C07183=1025.011,-6.218,-95.865,167.267,47.387,158.718
C07184=1025.005,-6.466,-95.851,167.264,47.390,158.718
C07185=1024.999,-6.717,-95.837,167.261,47.393,158.718
C07186=1024.992,-6.966,-95.824,167.259,47.397,158.718
C07187=1024.987,-7.216,-95.810,167.256,47.400,158.718
C07188=1024.980,-7.465,-95.796,167.254,47.403,158.719
C07189=1024.974,-7.714,-95.782,167.250,47.406,158.719
C07190=1024.967,-7.964,-95.768,167.248,47.410,158.719
C07191=1024.962,-8.214,-95.754,167.245,47.413,158.719
C07192=1024.956,-8.463,-95.741,167.242,47.416,158.720
C07193=1024.949,-8.713,-95.726,167.240,47.419,158.720
C07194=1024.943,-8.962,-95.713,167.237,47.422,158.720
C07195=1024.938,-9.212,-95.699,167.234,47.425,158.720
C07196=1024.932,-9.461,-95.685,167.232,47.428,158.721
C07197=1024.925,-9.711,-95.671,167.228,47.431,158.721
C07198=1024.920,-9.961,-95.658,167.227,47.435,158.721
C07199=1024.913,-10.210,-95.644,167.223,47.438,158.721
C07200=1024.907,-10.460,-95.629,167.221,47.441,158.721
C07201=1024.901,-10.709,-95.616,167.218,47.444,158.722
C07202=1024.896,-10.959,-95.602,167.215,47.448,158.722
C07203=1024.889,-11.209,-95.589,167.213,47.451,158.722
C07204=1024.883,-11.458,-95.575,167.210,47.454,158.722
C07205=1024.877,-11.707,-95.561,167.208,47.457,158.723
C07206=1024.872,-11.957,-95.548,167.204,47.460,158.723
C07207=1024.865,-12.207,-95.534,167.201,47.464,158.723
C07208=1024.859,-12.457,-95.520,167.199,47.466,158.723
C07209=1024.853,-12.705,-95.506,167.196,47.470,158.723
C07210=1024.847,-12.955,-95.492,167.194,47.472,158.724
C07211=1024.841,-13.205,-95.479,167.191,47.476,158.724
C07212=1024.835,-13.454,-95.465,167.189,47.479,158.724
C07213=1024.829,-13.704,-95.451,167.186,47.482,158.724
C07214=1024.823,-13.953,-95.438,167.182,47.485,158.725
C07215=1024.817,-14.202,-95.424,167.180,47.488,158.725
C07216=1024.811,-14.453,-95.410,167.177,47.491,158.725
C07217=1024.805,-14.702,-95.397,167.175,47.494,158.725
C07218=1024.799,-14.952,-95.383,167.172,47.497,158.725
C07219=1024.793,-15.201,-95.370,167.169,47.501,158.726
C07220=1024.787,-15.451,-95.355,167.167,47.504,158.726
C07221=1024.781,-15.700,-95.342,167.163,47.507,158.726
C07222=1024.775,-15.950,-95.329,167.161,47.510,158.726
C07223=1024.770,-16.200,-95.316,167.158,47.514,158.727
C07224=1024.763,-16.449,-95.303,167.155,47.517,158.727
C07225=1024.757,-16.699,-95.289,167.153,47.520,158.727
C07226=1024.750,-16.948,-95.276,167.150,47.523,158.727
C07227=1024.744,-17.198,-95.262,167.147,47.527,158.727
C07228=1024.739,-17.447,-95.248,167.145,47.530,158.728
C07229=1024.733,-17.697,-95.236,167.141,47.533,158.728
C07230=1024.726,-17.947,-95.222,167.138,47.537,158.728
C07231=1024.720,-18.196,-95.209,167.136,47.539,158.728
C07232=1024.714,-18.446,-95.195,167.133,47.543,158.729
C07233=1024.708,-18.695,-95.182,167.130,47.546,158.729
C07234=1024.702,-18.945,-95.169,167.128,47.549,158.729
C07235=1024.696,-19.194,-95.156,167.125,47.552,158.729
C07236=1024.690,-19.444,-95.142,167.122,47.555,158.729
C07237=1024.684,-19.694,-95.129,167.120,47.559,158.730
C07238=1024.677,-19.943,-95.115,167.117,47.562,158.730
C07239=1024.671,-20.193,-95.103,167.114,47.565,158.730
C07240=1024.665,-20.473,-95.087,167.110,47.569,158.730
C07241=1024.658,-20.753,-95.073,167.107,47.572,158.731
C07242=1024.651,-21.034,-95.058,167.104,47.576,158.731
C07243=1024.645,-21.315,-95.043,167.101,47.580,158.731
C07244=1024.639,-21.564,-95.030,167.098,47.583,158.731
C07245=1024.633,-21.813,-95.017,167.096,47.586,158.732
C07246=1024.626,-22.063,-95.003,167.093,47.589,158.732
C07247=1024.620,-22.313,-94.990,167.091,47.592,158.732
C07248=1024.614,-22.562,-94.977,167.088,47.596,158.732
C07249=1024.608,-22.812,-94.963,167.085,47.599,158.732
C07250=1024.602,-23.062,-94.951,167.082,47.602,158.733
C07251=1024.596,-23.311,-94.937,167.079,47.605,158.733
C07252=1024.591,-23.560,-94.924,167.076,47.609,158.733
C07253=1024.585,-23.810,-94.911,167.074,47.612,158.733
C07254=1024.578,-24.060,-94.898,167.071,47.615,158.733
C07255=1024.572,-24.309,-94.885,167.068,47.618,158.734
C07256=1024.566,-24.559,-94.872,167.066,47.621,158.734
C07257=1024.560,-24.808,-94.859,167.062,47.624,158.734
C07258=1024.555,-25.058,-94.846,167.059,47.628,158.734
C07259=1024.549,-25.307,-94.832,167.057,47.631,158.735
C07260=1024.543,-25.557,-94.820,167.054,47.634,158.735
C07261=1024.537,-25.807,-94.806,167.051,47.637,158.735
C07262=1024.530,-26.056,-94.793,167.049,47.640,158.735
C07263=1024.525,-26.306,-94.780,167.046,47.643,158.735
C07264=1024.519,-26.555,-94.767,167.044,47.646,158.736
C07265=1024.513,-26.805,-94.754,167.040,47.650,158.736
C07266=1024.507,-27.054,-94.741,167.037,47.653,158.736
C07267=1024.501,-27.304,-94.728,167.035,47.656,158.736
C07268=1024.495,-27.554,-94.715,167.032,47.659,158.736
C07269=1024.489,-27.804,-94.703,167.029,47.663,158.737
C07270=1024.483,-28.053,-94.689,167.026,47.666,158.737
C07271=1024.477,-28.303,-94.677,167.024,47.669,158.737
C07272=1024.471,-28.553,-94.664,167.021,47.672,158.737
C07273=1024.465,-28.802,-94.651,167.018,47.676,158.737
C07274=1024.459,-29.052,-94.638,167.015,47.678,158.738
C07275=1024.452,-29.301,-94.625,167.012,47.682,158.738
C07276=1024.447,-29.551,-94.613,167.009,47.685,158.738
C07277=1024.441,-29.801,-94.600,167.006,47.689,158.738
C07278=1024.434,-30.050,-94.587,167.004,47.691,158.738
C07279=1024.429,-30.300,-94.574,167.001,47.695,158.739
C07280=1024.423,-30.550,-94.562,166.998,47.698,158.739
C07281=1024.416,-30.799,-94.549,166.995,47.702,158.739
C07282=1024.410,-31.049,-94.536,166.992,47.704,158.739
C07283=1024.404,-31.298,-94.524,166.990,47.708,158.740
C07284=1024.398,-31.547,-94.511,166.986,47.711,158.740
C07285=1024.392,-31.797,-94.498,166.984,47.714,158.740
C07286=1024.386,-32.047,-94.486,166.981,47.718,158.740
C07287=1024.380,-32.296,-94.473,166.978,47.721,158.740
C07288=1024.374,-32.546,-94.460,166.975,47.724,158.741
C07289=1024.368,-32.796,-94.447,166.973,47.727,158.741
C07290=1024.362,-33.046,-94.435,166.970,47.731,158.741
C07291=1024.356,-33.295,-94.422,166.967,47.734,158.741
C07292=1024.350,-33.545,-94.410,166.964,47.737,158.741
C07293=1024.344,-33.794,-94.397,166.961,47.740,158.742
C07294=1024.338,-34.044,-94.385,166.958,47.744,158.742
C07295=1024.332,-34.293,-94.372,166.955,47.747,158.742
C07296=1024.326,-34.543,-94.359,166.953,47.750,158.742
C07297=1024.320,-34.793,-94.347,166.950,47.753,158.742
C07298=1024.314,-35.043,-94.334,166.947,47.757,158.743
C07299=1024.308,-35.292,-94.321,166.945,47.760,158.743
C07300=1024.303,-35.541,-94.309,166.942,47.763,158.743
C07301=1024.296,-35.791,-94.297,166.938,47.766,158.743
C07302=1024.290,-36.040,-94.284,166.935,47.770,158.743
C07303=1024.284,-36.290,-94.271,166.933,47.772,158.744
C07304=1024.278,-36.570,-94.257,166.930,47.776,158.744
C07305=1024.272,-36.849,-94.243,166.926,47.780,158.744
C07306=1024.265,-37.129,-94.230,166.923,47.784,158.744
C07307=1024.258,-37.408,-94.215,166.920,47.787,158.745
C07308=1024.252,-37.658,-94.203,166.917,47.791,158.745
C07309=1024.246,-37.908,-94.190,166.915,47.793,158.745
C07310=1024.241,-38.157,-94.178,166.912,47.797,158.745
C07311=1024.234,-38.407,-94.166,166.908,47.800,158.745
C07312=1024.228,-38.656,-94.153,166.905,47.803,158.745
C07313=1024.222,-38.906,-94.140,166.903,47.807,158.746
C07314=1024.216,-39.156,-94.128,166.900,47.810,158.746
C07315=1024.211,-39.405,-94.115,166.897,47.813,158.746
C07316=1024.204,-39.654,-94.103,166.894,47.816,158.746
C07317=1024.198,-39.904,-94.091,166.892,47.820,158.747
C07318=1024.193,-40.155,-94.079,166.889,47.823,158.747
C07319=1024.187,-40.404,-94.067,166.886,47.826,158.747
C07320=1024.181,-40.654,-94.055,166.883,47.830,158.747
C07321=1024.175,-40.903,-94.042,166.880,47.833,158.747
C07322=1024.168,-41.153,-94.030,166.877,47.836,158.748
C07323=1024.163,-41.402,-94.018,166.874,47.840,158.748
C07324=1024.156,-41.652,-94.006,166.871,47.843,158.748
C07325=1024.151,-41.902,-93.994,166.868,47.846,158.748
C07326=1024.145,-42.152,-93.981,166.866,47.850,158.748
C07327=1024.139,-42.400,-93.969,166.863,47.853,158.749
C07328=1024.133,-42.650,-93.957,166.860,47.856,158.749
C07329=1024.126,-42.900,-93.946,166.857,47.859,158.749
C07330=1024.121,-43.150,-93.933,166.854,47.863,158.749
C07331=1024.115,-43.400,-93.921,166.852,47.866,158.749
C07332=1024.108,-43.649,-93.909,166.848,47.869,158.750
C07333=1024.103,-43.899,-93.896,166.845,47.873,158.750
C07334=1024.097,-44.148,-93.885,166.842,47.876,158.750
C07335=1024.091,-44.398,-93.872,166.839,47.879,158.750
C07336=1024.085,-44.648,-93.860,166.837,47.882,158.750
C07337=1024.079,-44.897,-93.849,166.834,47.886,158.751
C07338=1024.073,-45.147,-93.836,166.831,47.889,158.751
C07339=1024.067,-45.396,-93.825,166.828,47.892,158.751
C07340=1024.061,-45.646,-93.812,166.825,47.895,158.751
C07341=1024.055,-45.896,-93.800,166.823,47.899,158.751
C07342=1024.049,-46.145,-93.789,166.819,47.902,158.752
C07343=1024.044,-46.395,-93.776,166.816,47.905,158.752
C07344=1024.037,-46.645,-93.764,166.813,47.909,158.752
C07345=1024.032,-46.894,-93.753,166.811,47.912,158.752
C07346=1024.026,-47.144,-93.740,166.808,47.915,158.752
C07347=1024.020,-47.393,-93.729,166.805,47.918,158.753
C07348=1024.014,-47.643,-93.716,166.802,47.922,158.753
C07349=1024.008,-47.893,-93.705,166.799,47.925,158.753
C07350=1024.002,-48.142,-93.693,166.797,47.928,158.753
C07351=1023.996,-48.392,-93.680,166.793,47.932,158.753
C07352=1023.991,-48.642,-93.669,166.790,47.935,158.753
C07353=1023.985,-48.892,-93.657,166.787,47.938,158.754
C07354=1023.978,-49.141,-93.645,166.785,47.941,158.754
C07355=1023.973,-49.391,-93.633,166.782,47.945,158.754
C07356=1023.967,-49.641,-93.621,166.779,47.948,158.754
C07357=1023.961,-49.890,-93.609,166.776,47.951,158.754
C07358=1023.956,-50.140,-93.597,166.773,47.954,158.755
C07359=1023.950,-50.389,-93.586,166.770,47.957,158.755
C07360=1023.944,-50.639,-93.573,166.767,47.961,158.755
C07361=1023.938,-50.889,-93.562,166.764,47.964,158.755
C07362=1023.931,-51.138,-93.550,166.761,47.967,158.755
C07363=1023.926,-51.389,-93.538,166.758,47.971,158.756
C07364=1023.920,-51.637,-93.527,166.755,47.974,158.756
C07365=1023.913,-51.888,-93.516,166.753,47.978,158.756
C07366=1023.908,-52.137,-93.505,166.750,47.981,158.756
C07367=1023.901,-52.387,-93.493,166.747,47.984,158.756
C07368=1023.894,-52.666,-93.480,166.743,47.988,158.757
C07369=1023.887,-52.947,-93.467,166.740,47.992,158.757
C07370=1023.881,-53.227,-93.454,166.737,47.996,158.757
C07371=1023.875,-53.507,-93.441,166.733,48.000,158.757
C07372=1023.869,-53.756,-93.430,166.730,48.004,158.757
C07373=1023.862,-54.006,-93.418,166.727,48.007,158.758
C07374=1023.856,-54.255,-93.407,166.725,48.010,158.758
C07375=1023.850,-54.505,-93.395,166.722,48.013,158.758
C07376=1023.844,-54.755,-93.385,166.719,48.017,158.758
C07377=1023.838,-55.005,-93.372,166.716,48.021,158.759
C07378=1023.833,-55.254,-93.361,166.713,48.024,158.759
C07379=1023.826,-55.504,-93.350,166.710,48.028,158.759
C07380=1023.820,-55.753,-93.338,166.706,48.031,158.759
C07381=1023.814,-56.003,-93.327,166.704,48.035,158.759
C07382=1023.809,-56.253,-93.316,166.700,48.038,158.760
C07383=1023.803,-56.502,-93.304,166.698,48.041,158.760
C07384=1023.796,-56.752,-93.293,166.695,48.045,158.760
C07385=1023.791,-57.002,-93.282,166.692,48.048,158.760
C07386=1023.784,-57.251,-93.270,166.689,48.052,158.760
C07387=1023.778,-57.501,-93.259,166.686,48.055,158.761
C07388=1023.773,-57.751,-93.247,166.683,48.058,158.761
C07389=1023.767,-58.001,-93.236,166.680,48.062,158.761
C07390=1023.761,-58.250,-93.225,166.677,48.065,158.761
C07391=1023.755,-58.500,-93.213,166.674,48.068,158.761
C07392=1023.749,-58.749,-93.203,166.672,48.072,158.762
C07393=1023.742,-58.999,-93.191,166.669,48.075,158.762
C07394=1023.737,-59.249,-93.180,166.666,48.079,158.762
C07395=1023.731,-59.498,-93.168,166.663,48.082,158.762
C07396=1023.725,-59.748,-93.157,166.659,48.085,158.762
C07397=1023.719,-59.998,-93.146,166.656,48.089,158.763
C07398=1023.714,-60.247,-93.135,166.653,48.092,158.763
C07399=1023.707,-60.497,-93.124,166.650,48.096,158.763
C07400=1023.701,-60.746,-93.112,166.647,48.099,158.763
C07401=1023.696,-60.996,-93.101,166.645,48.102,158.763
C07402=1023.690,-61.246,-93.090,166.642,48.106,158.764
C07403=1023.684,-61.496,-93.079,166.639,48.109,158.764
C07404=1023.678,-61.745,-93.068,166.636,48.113,158.764
C07405=1023.672,-61.995,-93.057,166.633,48.116,158.764
C07406=1023.666,-62.245,-93.046,166.629,48.119,158.764
C07407=1023.660,-62.494,-93.034,166.627,48.123,158.764
C07408=1023.655,-62.744,-93.022,166.623,48.126,158.765
///RCONF 1,0,0,1,0,0,0,0,0,0,0,0,0,0,0,0,0,0,0,0,0,0,0,0
C07409=1023.649,-62.994,-93.012,166.620,48.129,158.765
C07410=1023.643,-63.243,-93.001,166.618,48.133,158.765
C07411=1023.637,-63.494,-92.989,166.615,48.136,158.765
C07412=1023.631,-63.743,-92.979,166.612,48.139,158.765
C07413=1023.625,-63.992,-92.968,166.609,48.143,158.765
C07414=1023.620,-64.242,-92.957,166.606,48.146,158.766
C07415=1023.614,-64.492,-92.945,166.603,48.150,158.766
C07416=1023.608,-64.742,-92.934,166.600,48.153,158.766
C07417=1023.603,-64.991,-92.923,166.596,48.156,158.766
C07418=1023.597,-65.241,-92.912,166.595,48.160,158.767
C07419=1023.590,-65.491,-92.901,166.591,48.163,158.767
C07420=1023.585,-65.741,-92.890,166.588,48.166,158.767
C07421=1023.579,-65.990,-92.879,166.585,48.169,158.767
C07422=1023.573,-66.240,-92.868,166.582,48.173,158.767
C07423=1023.568,-66.489,-92.857,166.579,48.176,158.767
C07424=1023.562,-66.740,-92.846,166.576,48.180,158.767
C07425=1023.556,-66.989,-92.835,166.573,48.183,158.768
C07426=1023.550,-67.239,-92.824,166.571,48.186,158.768
C07427=1023.545,-67.488,-92.813,166.568,48.190,158.768
C07428=1023.539,-67.738,-92.802,166.564,48.193,158.768
C07429=1023.533,-67.988,-92.791,166.561,48.196,158.768
C07430=1023.527,-68.237,-92.780,166.558,48.200,158.769
C07431=1023.521,-68.487,-92.769,166.555,48.203,158.769
C07432=1023.516,-68.768,-92.757,166.552,48.206,158.769
C07433=1023.508,-69.049,-92.744,166.549,48.210,158.769
C07434=1023.502,-69.330,-92.733,166.545,48.214,158.769
C07435=1023.496,-69.612,-92.720,166.542,48.218,158.769
C07436=1023.490,-69.861,-92.709,166.539,48.221,158.770
C07437=1023.484,-70.111,-92.698,166.536,48.225,158.770
C07438=1023.479,-70.360,-92.687,166.533,48.228,158.770
C07439=1023.473,-70.610,-92.676,166.530,48.231,158.770
C07440=1023.467,-70.859,-92.666,166.528,48.234,158.770
C07441=1023.462,-71.109,-92.655,166.524,48.237,158.770
C07442=1023.456,-71.359,-92.644,166.522,48.241,158.771
C07443=1023.450,-71.609,-92.633,166.518,48.244,158.771
C07444=1023.444,-71.859,-92.622,166.515,48.247,158.771
C07445=1023.439,-72.108,-92.611,166.512,48.251,158.771
C07446=1023.433,-72.358,-92.600,166.509,48.254,158.771
C07447=1023.428,-72.608,-92.590,166.506,48.257,158.771
C07448=1023.422,-72.858,-92.579,166.504,48.261,158.772
C07449=1023.416,-73.107,-92.568,166.501,48.264,158.772
C07450=1023.411,-73.356,-92.557,166.497,48.267,158.772
C07451=1023.405,-73.606,-92.546,166.494,48.270,158.772
C07452=1023.399,-73.856,-92.536,166.491,48.274,158.772
C07453=1023.394,-74.106,-92.525,166.488,48.277,158.772
C07454=1023.388,-74.355,-92.514,166.485,48.281,158.773
C07455=1023.383,-74.605,-92.504,166.483,48.284,158.773
C07456=1023.377,-74.855,-92.493,166.480,48.287,158.773
C07457=1023.371,-75.105,-92.483,166.477,48.291,158.773
C07458=1023.365,-75.355,-92.472,166.474,48.294,158.773
C07459=1023.359,-75.604,-92.462,166.470,48.297,158.773
C07460=1023.353,-75.854,-92.452,166.468,48.301,158.774
C07461=1023.347,-76.104,-92.441,166.464,48.304,158.774
C07462=1023.342,-76.354,-92.431,166.461,48.307,158.774
C07463=1023.336,-76.603,-92.420,166.458,48.311,158.774
C07464=1023.330,-76.853,-92.410,166.455,48.315,158.774
C07465=1023.324,-77.103,-92.399,166.452,48.318,158.774
C07466=1023.319,-77.353,-92.389,166.449,48.322,158.775
C07467=1023.313,-77.602,-92.378,166.446,48.325,158.775
C07468=1023.307,-77.852,-92.369,166.443,48.328,158.775
C07469=1023.301,-78.102,-92.358,166.440,48.332,158.775
C07470=1023.296,-78.352,-92.348,166.437,48.335,158.775
C07471=1023.290,-78.601,-92.337,166.434,48.338,158.775
C07472=1023.285,-78.851,-92.327,166.431,48.342,158.776
C07473=1023.279,-79.100,-92.317,166.429,48.345,158.776
C07474=1023.273,-79.350,-92.306,166.425,48.349,158.776
C07475=1023.268,-79.599,-92.296,166.422,48.352,158.776
C07476=1023.262,-79.849,-92.285,166.419,48.356,158.776
C07477=1023.256,-80.099,-92.275,166.416,48.359,158.777
C07478=1023.250,-80.349,-92.265,166.413,48.362,158.777
C07479=1023.245,-80.599,-92.255,166.410,48.366,158.777
C07480=1023.238,-80.848,-92.244,166.407,48.369,158.777
C07481=1023.233,-81.098,-92.234,166.404,48.373,158.777
C07482=1023.227,-81.348,-92.225,166.401,48.376,158.777
C07483=1023.221,-81.597,-92.214,166.398,48.380,158.778
C07484=1023.215,-81.847,-92.204,166.395,48.383,158.778
C07485=1023.209,-82.097,-92.194,166.392,48.387,158.778
C07486=1023.203,-82.347,-92.185,166.389,48.391,158.778
C07487=1023.197,-82.597,-92.174,166.386,48.395,158.779
C07488=1023.192,-82.846,-92.165,166.383,48.398,158.779
C07489=1023.186,-83.096,-92.154,166.380,48.402,158.779
C07490=1023.180,-83.346,-92.145,166.377,48.405,158.779
C07491=1023.175,-83.595,-92.134,166.374,48.408,158.779
C07492=1023.168,-83.845,-92.124,166.371,48.412,158.779
C07493=1023.163,-84.095,-92.114,166.368,48.415,158.780
C07494=1023.157,-84.345,-92.105,166.365,48.419,158.780
C07495=1023.151,-84.595,-92.094,166.362,48.422,158.780
C07496=1023.145,-84.877,-92.083,166.358,48.427,158.780
C07497=1023.138,-85.161,-92.072,166.354,48.431,158.780
C07498=1023.132,-85.443,-92.060,166.351,48.435,158.781
C07499=1023.125,-85.727,-92.049,166.347,48.439,158.781
C07500=1023.119,-85.977,-92.040,166.344,48.442,158.781
C07501=1023.114,-86.227,-92.030,166.341,48.446,158.781
C07502=1023.108,-86.476,-92.020,166.338,48.449,158.781
C07503=1023.103,-86.726,-92.010,166.335,48.453,158.781
C07504=1023.096,-86.975,-92.000,166.332,48.457,158.782
C07505=1023.091,-87.225,-91.990,166.329,48.460,158.782
C07506=1023.084,-87.475,-91.980,166.326,48.464,158.782
C07507=1023.080,-87.725,-91.970,166.323,48.467,158.782
C07508=1023.073,-87.974,-91.961,166.320,48.470,158.782
C07509=1023.068,-88.225,-91.951,166.317,48.474,158.783
C07510=1023.062,-88.474,-91.941,166.314,48.477,158.783
C07511=1023.057,-88.724,-91.931,166.311,48.481,158.783
C07512=1023.051,-88.974,-91.922,166.307,48.484,158.783
C07513=1023.045,-89.224,-91.912,166.304,48.488,158.783
C07514=1023.039,-89.473,-91.902,166.301,48.492,158.783
C07515=1023.034,-89.723,-91.892,166.298,48.495,158.784
C07516=1023.028,-89.973,-91.883,166.295,48.498,158.784
C07517=1023.023,-90.223,-91.872,166.292,48.502,158.784
C07518=1023.017,-90.472,-91.863,166.289,48.505,158.784
C07519=1023.012,-90.722,-91.853,166.286,48.509,158.784
C07520=1023.006,-90.972,-91.844,166.283,48.512,158.784
C07521=1022.999,-91.222,-91.834,166.280,48.516,158.784
C07522=1022.995,-91.471,-91.824,166.277,48.520,158.785
C07523=1022.988,-91.721,-91.815,166.274,48.523,158.785
C07524=1022.983,-91.971,-91.804,166.271,48.526,158.785
C07525=1022.977,-92.220,-91.795,166.269,48.530,158.785
C07526=1022.972,-92.470,-91.785,166.266,48.533,158.785
C07527=1022.966,-92.720,-91.776,166.263,48.536,158.786
C07528=1022.961,-92.969,-91.766,166.260,48.540,158.786
C07529=1022.955,-93.219,-91.756,166.257,48.543,158.786
C07530=1022.949,-93.469,-91.746,166.253,48.547,158.786
C07531=1022.944,-93.718,-91.737,166.251,48.551,158.786
C07532=1022.938,-93.969,-91.728,166.247,48.554,158.786
C07533=1022.933,-94.218,-91.718,166.244,48.557,158.787
C07534=1022.927,-94.468,-91.709,166.241,48.561,158.787
C07535=1022.922,-94.718,-91.698,166.238,48.564,158.787
C07536=1022.916,-94.967,-91.689,166.235,48.567,158.787
C07537=1022.911,-95.217,-91.679,166.232,48.571,158.787
C07538=1022.905,-95.466,-91.670,166.229,48.575,158.787
C07539=1022.900,-95.717,-91.660,166.226,48.578,158.787
C07540=1022.894,-95.967,-91.651,166.223,48.582,158.788
C07541=1022.888,-96.216,-91.642,166.220,48.585,158.788
C07542=1022.883,-96.466,-91.631,166.217,48.588,158.788
C07543=1022.877,-96.715,-91.622,166.213,48.591,158.788
C07544=1022.872,-96.966,-91.613,166.211,48.595,158.788
C07545=1022.866,-97.215,-91.604,166.207,48.599,158.788
C07546=1022.861,-97.465,-91.593,166.204,48.602,158.789
C07547=1022.855,-97.714,-91.584,166.201,48.606,158.789
C07548=1022.850,-97.965,-91.575,166.198,48.609,158.789
C07549=1022.843,-98.214,-91.566,166.195,48.612,158.789
C07550=1022.839,-98.464,-91.556,166.192,48.616,158.789
C07551=1022.833,-98.714,-91.547,166.189,48.620,158.789
C07552=1022.827,-98.963,-91.538,166.186,48.623,158.790
C07553=1022.821,-99.213,-91.528,166.183,48.627,158.790
C07554=1022.816,-99.463,-91.520,166.180,48.631,158.790
C07555=1022.809,-99.713,-91.510,166.177,48.634,158.790
C07556=1022.805,-99.963,-91.501,166.174,48.638,158.790
C07557=1022.799,-100.212,-91.492,166.171,48.641,158.791
C07558=1022.793,-100.462,-91.483,166.168,48.645,158.791
C07559=1022.787,-100.712,-91.474,166.165,48.648,158.791
C07560=1022.781,-100.997,-91.462,166.161,48.653,158.791
C07561=1022.775,-101.282,-91.453,166.157,48.657,158.791
C07562=1022.769,-101.568,-91.442,166.154,48.661,158.791
C07563=1022.761,-101.853,-91.432,166.151,48.665,158.792
C07564=1022.757,-102.103,-91.423,166.147,48.668,158.792
C07565=1022.751,-102.353,-91.413,166.145,48.672,158.792
C07566=1022.745,-102.602,-91.405,166.141,48.675,158.792
C07567=1022.739,-102.852,-91.395,166.139,48.679,158.792
C07568=1022.734,-103.102,-91.387,166.135,48.683,158.792
C07569=1022.728,-103.351,-91.377,166.132,48.686,158.793
C07570=1022.723,-103.602,-91.369,166.129,48.690,158.793
C07571=1022.718,-103.851,-91.359,166.126,48.693,158.793
C07572=1022.712,-104.101,-91.350,166.123,48.697,158.793
C07573=1022.706,-104.350,-91.341,166.120,48.700,158.793
C07574=1022.701,-104.600,-91.332,166.117,48.704,158.794
C07575=1022.695,-104.850,-91.323,166.114,48.708,158.794
C07576=1022.690,-105.100,-91.314,166.111,48.711,158.794
C07577=1022.684,-105.350,-91.305,166.108,48.715,158.794
C07578=1022.678,-105.599,-91.296,166.105,48.718,158.794
C07579=1022.673,-105.849,-91.288,166.102,48.722,158.794
C07580=1022.667,-106.099,-91.277,166.099,48.725,158.795
C07581=1022.662,-106.349,-91.269,166.096,48.729,158.795
C07582=1022.656,-106.599,-91.260,166.093,48.732,158.795
C07583=1022.651,-106.848,-91.251,166.089,48.736,158.795
C07584=1022.646,-107.098,-91.242,166.086,48.740,158.795
C07585=1022.640,-107.348,-91.234,166.083,48.743,158.795
C07586=1022.634,-107.598,-91.225,166.080,48.747,158.795
C07587=1022.629,-107.847,-91.216,166.077,48.750,158.796
C07588=1022.623,-108.098,-91.207,166.074,48.754,158.796
C07589=1022.618,-108.347,-91.199,166.071,48.758,158.796
C07590=1022.612,-108.596,-91.189,166.068,48.762,158.796
C07591=1022.606,-108.847,-91.181,166.065,48.765,158.796
C07592=1022.601,-109.097,-91.172,166.062,48.769,158.797
C07593=1022.596,-109.346,-91.164,166.059,48.772,158.797
C07594=1022.590,-109.597,-91.155,166.056,48.776,158.797
C07595=1022.584,-109.845,-91.146,166.053,48.779,158.797
C07596=1022.578,-110.095,-91.138,166.050,48.783,158.797
C07597=1022.573,-110.345,-91.129,166.047,48.787,158.797
C07598=1022.567,-110.595,-91.120,166.044,48.791,158.798
C07599=1022.562,-110.845,-91.112,166.041,48.794,158.798
C07600=1022.557,-111.095,-91.103,166.038,48.798,158.798
C07601=1022.550,-111.345,-91.094,166.034,48.801,158.798
C07602=1022.545,-111.594,-91.085,166.031,48.805,158.798
C07603=1022.540,-111.844,-91.077,166.028,48.809,158.798
C07604=1022.535,-112.094,-91.068,166.025,48.812,158.799
C07605=1022.529,-112.344,-91.059,166.022,48.816,158.799
C07606=1022.524,-112.594,-91.051,166.019,48.820,158.799
C07607=1022.518,-112.844,-91.042,166.016,48.823,158.799
C07608=1022.512,-113.093,-91.035,166.013,48.827,158.799
C07609=1022.507,-113.343,-91.026,166.010,48.830,158.799
C07610=1022.501,-113.592,-91.017,166.007,48.834,158.800
C07611=1022.496,-113.842,-91.008,166.004,48.837,158.800
C07612=1022.490,-114.092,-91.000,166.001,48.841,158.800
C07613=1022.485,-114.342,-90.991,165.998,48.845,158.800
C07614=1022.480,-114.591,-90.983,165.995,48.848,158.800
C07615=1022.474,-114.842,-90.974,165.992,48.852,158.800
C07616=1022.468,-115.091,-90.966,165.989,48.855,158.801
C07617=1022.463,-115.341,-90.957,165.986,48.859,158.801
C07618=1022.457,-115.591,-90.949,165.983,48.863,158.801
C07619=1022.452,-115.840,-90.940,165.979,48.867,158.801
C07620=1022.447,-116.091,-90.933,165.976,48.871,158.801
C07621=1022.441,-116.341,-90.924,165.973,48.874,158.801
C07622=1022.435,-116.590,-90.916,165.970,48.878,158.802
C07623=1022.430,-116.840,-90.907,165.967,48.881,158.802
C07624=1022.424,-117.125,-90.898,165.964,48.885,158.802
C07625=1022.418,-117.410,-90.888,165.960,48.889,158.802
C07626=1022.411,-117.695,-90.879,165.956,48.894,158.802
C07627=1022.405,-117.980,-90.869,165.953,48.898,158.803
C07628=1022.400,-118.229,-90.861,165.951,48.902,158.803
C07629=1022.394,-118.480,-90.853,165.946,48.905,158.803
C07630=1022.388,-118.730,-90.845,165.944,48.909,158.803
C07631=1022.383,-118.980,-90.836,165.940,48.913,158.803
C07632=1022.378,-119.229,-90.828,165.938,48.917,158.803
C07633=1022.372,-119.479,-90.819,165.934,48.920,158.804
C07634=1022.366,-119.728,-90.811,165.932,48.924,158.804
C07635=1022.361,-119.979,-90.804,165.928,48.927,158.804
C07636=1022.356,-120.228,-90.795,165.926,48.931,158.804
C07637=1022.350,-120.478,-90.787,165.922,48.934,158.804
C07638=1022.345,-120.727,-90.779,165.920,48.938,158.804
C07639=1022.340,-120.977,-90.770,165.917,48.942,158.805
C07640=1022.335,-121.228,-90.762,165.914,48.946,158.805
C07641=1022.329,-121.477,-90.755,165.911,48.950,158.805
C07642=1022.323,-121.727,-90.746,165.908,48.953,158.805
C07643=1022.318,-121.977,-90.738,165.905,48.957,158.805
C07644=1022.312,-122.226,-90.730,165.902,48.960,158.806
C07645=1022.307,-122.476,-90.722,165.898,48.964,158.806
C07646=1022.302,-122.726,-90.713,165.895,48.968,158.806
C07647=1022.296,-122.976,-90.706,165.892,48.972,158.806
C07648=1022.291,-123.226,-90.698,165.889,48.975,158.806
C07649=1022.286,-123.475,-90.689,165.886,48.979,158.806
C07650=1022.280,-123.725,-90.682,165.883,48.982,158.806
C07651=1022.275,-123.975,-90.674,165.880,48.986,158.807
C07652=1022.269,-124.225,-90.665,165.877,48.989,158.807
C07653=1022.264,-124.475,-90.658,165.874,48.993,158.807
C07654=1022.259,-124.724,-90.650,165.871,48.997,158.807
C07655=1022.253,-124.975,-90.642,165.868,49.001,158.807
C07656=1022.248,-125.224,-90.634,165.865,49.004,158.807
C07657=1022.242,-125.474,-90.625,165.862,49.008,158.808
C07658=1022.237,-125.724,-90.618,165.859,49.012,158.808
C07659=1022.231,-125.974,-90.610,165.855,49.016,158.808
C07660=1022.226,-126.224,-90.603,165.852,49.020,158.808
C07661=1022.220,-126.473,-90.594,165.849,49.023,158.808
C07662=1022.215,-126.723,-90.587,165.846,49.027,158.809
C07663=1022.209,-126.973,-90.578,165.843,49.031,158.809
C07664=1022.204,-127.223,-90.571,165.840,49.034,158.809
C07665=1022.198,-127.473,-90.563,165.837,49.038,158.809
C07666=1022.193,-127.723,-90.556,165.834,49.041,158.809
C07667=1022.188,-127.972,-90.547,165.831,49.045,158.809
C07668=1022.183,-128.222,-90.539,165.828,49.049,158.810
C07669=1022.178,-128.471,-90.531,165.825,49.051,158.809
C07670=1022.174,-128.721,-90.521,165.822,49.054,158.809
C07671=1022.170,-128.971,-90.511,165.820,49.056,158.809
C07672=1022.168,-129.220,-90.500,165.817,49.057,158.809
C07673=1022.165,-129.469,-90.490,165.815,49.058,158.809
C07674=1022.163,-129.719,-90.478,165.812,49.058,158.809
C07675=1022.161,-129.969,-90.465,165.809,49.058,158.808
C07676=1022.160,-130.219,-90.453,165.807,49.057,158.808
C07677=1022.160,-130.469,-90.439,165.805,49.056,158.807
C07678=1022.159,-130.719,-90.425,165.803,49.054,158.807
C07679=1022.160,-130.968,-90.410,165.801,49.052,158.806
C07680=1022.160,-131.219,-90.396,165.798,49.050,158.805
C07681=1022.162,-131.469,-90.379,165.797,49.046,158.804
C07682=1022.164,-131.718,-90.363,165.795,49.042,158.803
C07683=1022.166,-131.967,-90.346,165.793,49.038,158.802
C07684=1022.170,-132.218,-90.329,165.792,49.033,158.801
///RCONF 1,0,0,0,0,0,0,0,0,0,0,0,0,0,0,0,0,0,0,0,0,0,0,0
C07685=1022.172,-132.467,-90.310,165.790,49.028,158.800
C07686=1022.177,-132.717,-90.292,165.788,49.022,158.799
C07687=1022.181,-132.966,-90.273,165.786,49.016,158.798
C07688=1021.894,-132.993,-90.621,165.740,49.314,158.841
C07689=1021.889,-132.743,-90.640,165.742,49.320,158.842
C07690=1021.885,-132.493,-90.660,165.743,49.325,158.843
C07691=1021.882,-132.243,-90.677,165.744,49.331,158.845
C07692=1021.880,-131.993,-90.695,165.746,49.336,158.846
C07693=1021.877,-131.744,-90.712,165.748,49.340,158.847
C07694=1021.875,-131.494,-90.728,165.750,49.344,158.848
C07695=1021.874,-131.244,-90.744,165.752,49.346,158.848
C07696=1021.873,-130.994,-90.760,165.753,49.349,158.849
C07697=1021.873,-130.744,-90.775,165.756,49.352,158.850
C07698=1021.872,-130.495,-90.788,165.758,49.354,158.850
C07699=1021.874,-130.245,-90.801,165.761,49.355,158.851
C07700=1021.874,-129.995,-90.815,165.763,49.355,158.851
C07701=1021.876,-129.746,-90.827,165.765,49.355,158.852
C07702=1021.878,-129.496,-90.838,165.768,49.355,158.852
C07703=1021.880,-129.246,-90.849,165.770,49.355,158.852
C07704=1021.883,-128.996,-90.860,165.773,49.353,158.853
C07705=1021.887,-128.747,-90.870,165.775,49.351,158.853
C07706=1021.891,-128.497,-90.880,165.779,49.349,158.853
C07707=1021.895,-128.248,-90.888,165.781,49.346,158.853
C07708=1021.901,-127.998,-90.897,165.784,49.342,158.853
C07709=1021.905,-127.748,-90.905,165.787,49.339,158.853
C07710=1021.911,-127.499,-90.912,165.790,49.335,158.852
C07711=1021.916,-127.249,-90.920,165.793,49.331,158.852
C07712=1021.922,-127.000,-90.928,165.797,49.328,158.852
C07713=1021.927,-126.749,-90.935,165.800,49.323,158.852
C07714=1021.933,-126.500,-90.943,165.803,49.319,158.852
C07715=1021.938,-126.250,-90.951,165.806,49.316,158.852
C07716=1021.944,-126.000,-90.959,165.809,49.312,158.851
C07717=1021.949,-125.750,-90.967,165.812,49.309,158.851
C07718=1021.955,-125.500,-90.975,165.815,49.305,158.851
C07719=1021.960,-125.250,-90.982,165.817,49.301,158.851
C07720=1021.966,-125.001,-90.990,165.821,49.297,158.851
C07721=1021.971,-124.750,-90.998,165.824,49.293,158.850
C07722=1021.977,-124.501,-91.006,165.827,49.289,158.850
C07723=1021.981,-124.252,-91.014,165.830,49.286,158.850
C07724=1021.986,-124.002,-91.022,165.833,49.282,158.850
C07725=1021.992,-123.752,-91.030,165.836,49.278,158.850
C07726=1021.997,-123.502,-91.038,165.839,49.274,158.850
C07727=1022.003,-123.252,-91.046,165.842,49.271,158.849
C07728=1022.009,-123.003,-91.054,165.845,49.267,158.849
C07729=1022.013,-122.752,-91.062,165.848,49.263,158.849
C07730=1022.019,-122.503,-91.070,165.852,49.260,158.849
C07731=1022.025,-122.253,-91.078,165.855,49.256,158.849
C07732=1022.030,-122.003,-91.086,165.858,49.252,158.849
C07733=1022.035,-121.753,-91.094,165.861,49.248,158.848
C07734=1022.040,-121.503,-91.103,165.864,49.245,158.848
C07735=1022.046,-121.254,-91.111,165.867,49.241,158.848
C07736=1022.051,-121.004,-91.118,165.869,49.237,158.848
C07737=1022.056,-120.754,-91.127,165.872,49.234,158.848
C07738=1022.062,-120.505,-91.135,165.875,49.230,158.847
C07739=1022.068,-120.255,-91.143,165.878,49.226,158.847
C07740=1022.073,-120.005,-91.151,165.882,49.222,158.847
C07741=1022.079,-119.754,-91.159,165.885,49.219,158.847
C07742=1022.085,-119.505,-91.168,165.888,49.215,158.847
C07743=1022.090,-119.255,-91.176,165.891,49.211,158.847
C07744=1022.095,-119.005,-91.184,165.894,49.207,158.847
C07745=1022.101,-118.755,-91.192,165.897,49.203,158.846
C07746=1022.106,-118.506,-91.200,165.900,49.200,158.846
C07747=1022.111,-118.256,-91.209,165.903,49.196,158.846
C07748=1022.117,-118.006,-91.217,165.906,49.192,158.846
C07749=1022.123,-117.721,-91.227,165.910,49.188,158.846
C07750=1022.129,-117.436,-91.236,165.913,49.183,158.845
C07751=1022.135,-117.151,-91.245,165.916,49.179,158.845
C07752=1022.141,-116.866,-91.255,165.920,49.175,158.845
C07753=1022.147,-116.617,-91.263,165.923,49.172,158.845
C07754=1022.153,-116.367,-91.271,165.926,49.168,158.845
C07755=1022.158,-116.117,-91.280,165.929,49.164,158.844
C07756=1022.164,-115.867,-91.289,165.933,49.160,158.844
C07757=1022.169,-115.617,-91.297,165.936,49.156,158.844
C07758=1022.175,-115.368,-91.305,165.939,49.153,158.844
C07759=1022.180,-115.118,-91.313,165.942,49.149,158.844
C07760=1022.185,-114.868,-91.322,165.945,49.146,158.844
C07761=1022.191,-114.619,-91.330,165.948,49.142,158.843
C07762=1022.197,-114.368,-91.339,165.950,49.138,158.843
C07763=1022.203,-114.119,-91.347,165.954,49.134,158.843
C07764=1022.208,-113.869,-91.356,165.956,49.130,158.843
C07765=1022.213,-113.619,-91.364,165.961,49.127,158.843
C07766=1022.218,-113.370,-91.373,165.963,49.123,158.843
C07767=1022.224,-113.119,-91.381,165.967,49.119,158.843
C07768=1022.230,-112.869,-91.390,165.969,49.115,158.842
C07769=1022.235,-112.620,-91.398,165.973,49.112,158.842
C07770=1022.240,-112.370,-91.407,165.975,49.108,158.842
C07771=1022.245,-112.120,-91.415,165.978,49.105,158.842
C07772=1022.251,-111.870,-91.424,165.981,49.101,158.842
C07773=1022.256,-111.620,-91.433,165.984,49.098,158.841
C07774=1022.262,-111.370,-91.441,165.987,49.094,158.841
C07775=1022.268,-111.121,-91.449,165.990,49.090,158.841
C07776=1022.274,-110.871,-91.459,165.994,49.086,158.841
C07777=1022.279,-110.622,-91.467,165.997,49.082,158.841
C07778=1022.284,-110.372,-91.476,166.000,49.079,158.841
C07779=1022.290,-110.122,-91.484,166.003,49.075,158.840
C07780=1022.296,-109.872,-91.493,166.006,49.071,158.840
C07781=1022.301,-109.622,-91.502,166.009,49.067,158.840
C07782=1022.306,-109.373,-91.511,166.012,49.064,158.840
C07783=1022.312,-109.123,-91.519,166.015,49.060,158.840
C07784=1022.318,-108.873,-91.528,166.018,49.056,158.839
C07785=1022.323,-108.623,-91.537,166.021,49.053,158.839
C07786=1022.328,-108.373,-91.545,166.025,49.049,158.839
C07787=1022.334,-108.123,-91.555,166.028,49.045,158.839
C07788=1022.339,-107.874,-91.563,166.031,49.041,158.839
C07789=1022.345,-107.624,-91.572,166.034,49.038,158.839
C07790=1022.351,-107.374,-91.580,166.037,49.034,158.838
C07791=1022.356,-107.125,-91.590,166.040,49.031,158.838
C07792=1022.361,-106.875,-91.598,166.043,49.027,158.838
C07793=1022.367,-106.624,-91.607,166.046,49.023,158.838
C07794=1022.373,-106.375,-91.615,166.049,49.019,158.838
C07795=1022.378,-106.126,-91.625,166.052,49.016,158.838
C07796=1022.384,-105.875,-91.633,166.054,49.012,158.837
C07797=1022.390,-105.626,-91.643,166.059,49.009,158.837
C07798=1022.395,-105.376,-91.651,166.061,49.005,158.837
C07799=1022.401,-105.126,-91.660,166.065,49.001,158.837
C07800=1022.406,-104.877,-91.669,166.067,48.997,158.837
C07801=1022.411,-104.626,-91.679,166.071,48.994,158.837
C07802=1022.417,-104.376,-91.687,166.073,48.990,158.836
C07803=1022.422,-104.127,-91.696,166.077,48.987,158.836
C07804=1022.428,-103.877,-91.705,166.079,48.983,158.836
C07805=1022.434,-103.628,-91.714,166.083,48.980,158.836
C07806=1022.440,-103.377,-91.723,166.085,48.976,158.836
C07807=1022.445,-103.128,-91.732,166.088,48.972,158.836
C07808=1022.450,-102.879,-91.741,166.091,48.968,158.835
C07809=1022.455,-102.628,-91.750,166.094,48.965,158.835
C07810=1022.461,-102.379,-91.760,166.097,48.961,158.835
C07811=1022.467,-102.128,-91.768,166.101,48.957,158.835
C07812=1022.473,-101.879,-91.778,166.104,48.954,158.835
C07813=1022.479,-101.593,-91.788,166.107,48.950,158.834
C07814=1022.485,-101.309,-91.798,166.111,48.945,158.834
C07815=1022.491,-101.023,-91.809,166.115,48.941,158.834
C07816=1022.498,-100.738,-91.820,166.118,48.937,158.834
C07817=1022.504,-100.489,-91.828,166.121,48.934,158.834
C07818=1022.510,-100.239,-91.838,166.124,48.930,158.833
C07819=1022.514,-99.989,-91.847,166.128,48.926,158.833
C07820=1022.521,-99.739,-91.856,166.131,48.922,158.833
C07821=1022.526,-99.490,-91.865,166.134,48.919,158.833
C07822=1022.532,-99.239,-91.874,166.137,48.915,158.833
C07823=1022.538,-98.990,-91.883,166.140,48.912,158.833
C07824=1022.543,-98.740,-91.892,166.143,48.908,158.832
C07825=1022.548,-98.490,-91.902,166.145,48.904,158.832
C07826=1022.554,-98.241,-91.912,166.148,48.900,158.832
C07827=1022.560,-97.991,-91.920,166.151,48.896,158.832
C07828=1022.566,-97.741,-91.930,166.154,48.893,158.832
C07829=1022.571,-97.492,-91.940,166.157,48.889,158.831
C07830=1022.577,-97.241,-91.948,166.160,48.886,158.831
C07831=1022.582,-96.992,-91.958,166.164,48.883,158.831
C07832=1022.588,-96.742,-91.968,166.166,48.879,158.831
C07833=1022.593,-96.493,-91.977,166.170,48.875,158.831
C07834=1022.598,-96.242,-91.986,166.173,48.872,158.831
C07835=1022.604,-95.993,-91.996,166.176,48.868,158.831
C07836=1022.609,-95.743,-92.006,166.179,48.865,158.830
C07837=1022.615,-95.493,-92.015,166.182,48.862,158.830
C07838=1022.621,-95.244,-92.025,166.185,48.858,158.830
C07839=1022.626,-94.993,-92.034,166.188,48.854,158.830
C07840=1022.632,-94.744,-92.043,166.191,48.851,158.830
C07841=1022.637,-94.494,-92.053,166.195,48.847,158.830
C07842=1022.643,-94.245,-92.063,166.198,48.844,158.830
C07843=1022.648,-93.995,-92.073,166.201,48.840,158.829
C07844=1022.654,-93.745,-92.082,166.204,48.836,158.829
C07845=1022.659,-93.495,-92.091,166.207,48.833,158.829
C07846=1022.665,-93.245,-92.101,166.210,48.829,158.829
C07847=1022.671,-92.996,-92.110,166.213,48.826,158.829
C07848=1022.676,-92.746,-92.120,166.216,48.822,158.828
C07849=1022.682,-92.496,-92.130,166.219,48.819,158.828
C07850=1022.687,-92.247,-92.140,166.222,48.815,158.828
C07851=1022.693,-91.997,-92.149,166.225,48.812,158.828
C07852=1022.699,-91.747,-92.159,166.228,48.808,158.828
C07853=1022.704,-91.498,-92.169,166.231,48.804,158.828
C07854=1022.710,-91.248,-92.179,166.234,48.801,158.828
C07855=1022.716,-90.998,-92.188,166.237,48.797,158.827
C07856=1022.721,-90.749,-92.198,166.240,48.794,158.827
C07857=1022.727,-90.498,-92.207,166.243,48.790,158.827
C07858=1022.732,-90.248,-92.217,166.246,48.787,158.827
C07859=1022.738,-89.999,-92.226,166.249,48.783,158.827
C07860=1022.744,-89.749,-92.236,166.252,48.779,158.826
C07861=1022.749,-89.499,-92.246,166.255,48.776,158.826
C07862=1022.755,-89.249,-92.256,166.258,48.772,158.826
C07863=1022.760,-89.000,-92.265,166.261,48.769,158.826
C07864=1022.766,-88.750,-92.275,166.264,48.765,158.826
C07865=1022.772,-88.501,-92.286,166.267,48.762,158.826
C07866=1022.778,-88.251,-92.295,166.270,48.758,158.825
C07867=1022.783,-88.002,-92.305,166.273,48.754,158.825
C07868=1022.789,-87.752,-92.315,166.276,48.751,158.825
C07869=1022.795,-87.502,-92.325,166.279,48.747,158.825
C07870=1022.801,-87.252,-92.334,166.282,48.744,158.825
C07871=1022.806,-87.002,-92.344,166.286,48.740,158.824
C07872=1022.812,-86.753,-92.354,166.289,48.737,158.824
C07873=1022.817,-86.502,-92.364,166.292,48.733,158.824
C07874=1022.823,-86.253,-92.374,166.295,48.729,158.824
C07875=1022.828,-86.003,-92.383,166.298,48.725,158.824
C07876=1022.834,-85.753,-92.393,166.301,48.722,158.824
C07877=1022.842,-85.470,-92.405,166.304,48.718,158.823
C07878=1022.847,-85.187,-92.416,166.308,48.714,158.823
C07879=1022.854,-84.904,-92.428,166.312,48.710,158.823
C07880=1022.861,-84.621,-92.438,166.315,48.706,158.823
C07881=1022.866,-84.371,-92.448,166.318,48.702,158.822
C07882=1022.872,-84.121,-92.458,166.321,48.699,158.822
C07883=1022.878,-83.871,-92.468,166.324,48.695,158.822
C07884=1022.884,-83.622,-92.478,166.327,48.691,158.822
C07885=1022.890,-83.372,-92.488,166.329,48.687,158.822
C07886=1022.895,-83.123,-92.498,166.334,48.684,158.822
C07887=1022.901,-82.873,-92.508,166.337,48.680,158.821
C07888=1022.907,-82.623,-92.517,166.340,48.677,158.821
C07889=1022.912,-82.374,-92.528,166.343,48.673,158.821
C07890=1022.919,-82.124,-92.538,166.346,48.669,158.821
C07891=1022.924,-81.874,-92.548,166.348,48.666,158.821
C07892=1022.930,-81.624,-92.558,166.351,48.662,158.820
C07893=1022.936,-81.374,-92.568,166.354,48.658,158.820
C07894=1022.942,-81.125,-92.578,166.357,48.654,158.820
C07895=1022.947,-80.875,-92.588,166.360,48.651,158.820
C07896=1022.953,-80.626,-92.598,166.363,48.647,158.820
C07897=1022.959,-80.376,-92.608,166.366,48.644,158.819
C07898=1022.965,-80.126,-92.618,166.369,48.640,158.819
C07899=1022.971,-79.877,-92.629,166.372,48.637,158.819
C07900=1022.976,-79.626,-92.639,166.375,48.633,158.819
C07901=1022.982,-79.376,-92.649,166.378,48.630,158.819
C07902=1022.988,-79.127,-92.659,166.382,48.626,158.819
C07903=1022.994,-78.877,-92.669,166.384,48.622,158.818
C07904=1022.999,-78.628,-92.680,166.388,48.619,158.818
C07905=1023.005,-78.377,-92.691,166.390,48.615,158.818
C07906=1023.010,-78.128,-92.701,166.394,48.612,158.818
C07907=1023.017,-77.878,-92.711,166.397,48.609,158.818
C07908=1023.022,-77.629,-92.722,166.400,48.605,158.817
C07909=1023.028,-77.379,-92.732,166.403,48.602,158.817
C07910=1023.034,-77.129,-92.743,166.406,48.598,158.817
C07911=1023.040,-76.879,-92.752,166.409,48.594,158.817
C07912=1023.045,-76.630,-92.763,166.412,48.591,158.817
C07913=1023.051,-76.380,-92.773,166.415,48.587,158.816
C07914=1023.057,-76.130,-92.784,166.418,48.584,158.816
C07915=1023.062,-75.880,-92.795,166.421,48.580,158.816
C07916=1023.069,-75.631,-92.805,166.424,48.577,158.816
C07917=1023.074,-75.381,-92.815,166.427,48.574,158.816
C07918=1023.080,-75.131,-92.826,166.430,48.570,158.816
C07919=1023.085,-74.881,-92.836,166.433,48.566,158.815
C07920=1023.091,-74.632,-92.847,166.436,48.562,158.815
C07921=1023.097,-74.383,-92.857,166.439,48.559,158.815
C07922=1023.103,-74.132,-92.867,166.442,48.556,158.815
C07923=1023.108,-73.883,-92.879,166.445,48.552,158.815
C07924=1023.114,-73.633,-92.890,166.448,48.549,158.815
C07925=1023.119,-73.383,-92.900,166.451,48.546,158.814
C07926=1023.125,-73.134,-92.911,166.455,48.542,158.814
C07927=1023.130,-72.884,-92.922,166.457,48.538,158.814
C07928=1023.136,-72.635,-92.932,166.460,48.535,158.814
C07929=1023.142,-72.384,-92.943,166.463,48.532,158.814
C07930=1023.147,-72.135,-92.953,166.466,48.529,158.814
C07931=1023.153,-71.886,-92.964,166.469,48.525,158.813
C07932=1023.159,-71.636,-92.975,166.472,48.522,158.813
C07933=1023.164,-71.386,-92.985,166.475,48.519,158.813
C07934=1023.169,-71.136,-92.997,166.478,48.515,158.813
C07935=1023.175,-70.887,-93.008,166.481,48.511,158.813
C07936=1023.181,-70.636,-93.019,166.484,48.508,158.813
C07937=1023.187,-70.387,-93.030,166.487,48.505,158.812
C07938=1023.193,-70.137,-93.041,166.490,48.502,158.812
C07939=1023.198,-69.887,-93.051,166.492,48.498,158.812
C07940=1023.204,-69.638,-93.062,166.495,48.495,158.812
C07941=1023.211,-69.358,-93.074,166.499,48.491,158.812
C07942=1023.217,-69.076,-93.087,166.502,48.487,158.812
C07943=1023.223,-68.795,-93.098,166.506,48.483,158.811
C07944=1023.230,-68.514,-93.111,166.509,48.479,158.811
C07945=1023.235,-68.265,-93.122,166.512,48.476,158.811
C07946=1023.242,-68.015,-93.133,166.516,48.473,158.811
C07947=1023.247,-67.765,-93.144,166.518,48.469,158.811
C07948=1023.252,-67.515,-93.155,166.522,48.466,158.810
C07949=1023.258,-67.265,-93.166,166.525,48.463,158.810
C07950=1023.264,-67.016,-93.176,166.528,48.459,158.810
C07951=1023.269,-66.766,-93.187,166.530,48.456,158.810
C07952=1023.276,-66.516,-93.199,166.533,48.452,158.810
C07953=1023.281,-66.267,-93.209,166.536,48.449,158.809
C07954=1023.287,-66.017,-93.220,166.539,48.445,158.809
C07955=1023.293,-65.768,-93.231,166.542,48.442,158.809
C07956=1023.299,-65.518,-93.242,166.545,48.438,158.809
C07957=1023.304,-65.268,-93.254,166.548,48.435,158.809
C07958=1023.310,-65.018,-93.265,166.551,48.432,158.809
C07959=1023.316,-64.769,-93.276,166.554,48.428,158.808
C07960=1023.321,-64.519,-93.286,166.557,48.425,158.808
C07961=1023.328,-64.269,-93.298,166.560,48.421,158.808
C07962=1023.334,-64.019,-93.309,166.563,48.417,158.808
C07963=1023.339,-63.770,-93.319,166.566,48.414,158.808
C07964=1023.345,-63.520,-93.330,166.569,48.410,158.807
C07965=1023.351,-63.270,-93.342,166.571,48.407,158.807
C07966=1023.356,-63.020,-93.353,166.575,48.404,158.807
C07967=1023.362,-62.772,-93.365,166.577,48.400,158.807
///RCONF 1,0,0,1,0,0,0,0,0,0,0,0,0,0,0,0,0,0,0,0,0,0,0,0
C07968=1023.368,-62.522,-93.376,166.581,48.397,158.807
C07969=1023.375,-62.272,-93.387,166.584,48.394,158.807
C07970=1023.380,-62.022,-93.398,166.587,48.390,158.806
C07971=1023.386,-61.773,-93.409,166.590,48.387,158.806
C07972=1023.392,-61.522,-93.420,166.593,48.383,158.806
C07973=1023.397,-61.273,-93.431,166.596,48.380,158.806
C07974=1023.403,-61.023,-93.442,166.599,48.376,158.806
C07975=1023.409,-60.773,-93.453,166.602,48.372,158.805
C07976=1023.415,-60.524,-93.464,166.605,48.369,158.805
C07977=1023.421,-60.275,-93.476,166.608,48.365,158.805
C07978=1023.428,-60.025,-93.487,166.611,48.362,158.805
C07979=1023.433,-59.775,-93.499,166.614,48.358,158.804
C07980=1023.438,-59.525,-93.509,166.616,48.355,158.804
C07981=1023.445,-59.275,-93.521,166.619,48.352,158.804
C07982=1023.451,-59.026,-93.532,166.622,48.348,158.804
C07983=1023.456,-58.777,-93.543,166.625,48.345,158.804
C07984=1023.463,-58.527,-93.554,166.628,48.341,158.803
C07985=1023.468,-58.277,-93.566,166.631,48.338,158.803
C07986=1023.473,-58.027,-93.577,166.634,48.334,158.803
C07987=1023.480,-57.778,-93.589,166.637,48.331,158.803
C07988=1023.486,-57.528,-93.600,166.640,48.327,158.803
C07989=1023.492,-57.278,-93.611,166.643,48.324,158.802
C07990=1023.498,-57.029,-93.622,166.646,48.320,158.802
C07991=1023.503,-56.779,-93.634,166.649,48.316,158.802
C07992=1023.510,-56.529,-93.645,166.652,48.313,158.802
C07993=1023.515,-56.280,-93.656,166.655,48.309,158.802
C07994=1023.522,-56.030,-93.667,166.658,48.306,158.802
C07995=1023.528,-55.781,-93.679,166.661,48.302,158.801
C07996=1023.534,-55.531,-93.690,166.664,48.299,158.801
C07997=1023.539,-55.281,-93.702,166.667,48.295,158.801
C07998=1023.545,-55.032,-93.713,166.669,48.292,158.801
C07999=1023.551,-54.782,-93.724,166.672,48.288,158.800
C08000=1023.557,-54.532,-93.735,166.675,48.285,158.800
C08001=1023.564,-54.283,-93.747,166.678,48.281,158.800
C08002=1023.570,-54.033,-93.758,166.681,48.278,158.800
C08003=1023.575,-53.783,-93.770,166.684,48.274,158.799
C08004=1023.581,-53.534,-93.782,166.687,48.271,158.799
C08005=1023.588,-53.253,-93.794,166.691,48.267,158.799
C08006=1023.595,-52.974,-93.807,166.694,48.263,158.799
C08007=1023.602,-52.694,-93.820,166.697,48.259,158.799
C08008=1023.608,-52.414,-93.833,166.701,48.255,158.798
C08009=1023.615,-52.164,-93.844,166.704,48.251,158.798
C08010=1023.621,-51.915,-93.855,166.707,48.248,158.798
C08011=1023.627,-51.665,-93.867,166.710,48.244,158.798
C08012=1023.632,-51.415,-93.879,166.713,48.240,158.797
C08013=1023.639,-51.165,-93.890,166.716,48.237,158.797
C08014=1023.645,-50.916,-93.902,166.719,48.233,158.797
C08015=1023.651,-50.666,-93.913,166.721,48.230,158.797
C08016=1023.656,-50.417,-93.925,166.724,48.227,158.797
C08017=1023.662,-50.167,-93.938,166.727,48.223,158.796
C08018=1023.668,-49.918,-93.948,166.730,48.220,158.796
C08019=1023.674,-49.668,-93.961,166.733,48.216,158.796
C08020=1023.680,-49.418,-93.972,166.736,48.213,158.796
C08021=1023.685,-49.168,-93.984,166.738,48.210,158.796
C08022=1023.692,-48.919,-93.996,166.742,48.207,158.796
C08023=1023.697,-48.669,-94.008,166.745,48.203,158.795
C08024=1023.703,-48.419,-94.020,166.748,48.200,158.795
C08025=1023.709,-48.170,-94.032,166.751,48.197,158.795
C08026=1023.715,-47.920,-94.044,166.754,48.193,158.795
C08027=1023.721,-47.671,-94.055,166.756,48.190,158.794
C08028=1023.727,-47.421,-94.068,166.759,48.187,158.794
C08029=1023.733,-47.172,-94.080,166.762,48.183,158.794
C08030=1023.738,-46.922,-94.091,166.765,48.180,158.794
C08031=1023.744,-46.672,-94.104,166.768,48.176,158.794
C08032=1023.750,-46.423,-94.116,166.771,48.173,158.793
C08033=1023.756,-46.172,-94.127,166.773,48.170,158.793
C08034=1023.762,-45.923,-94.139,166.776,48.166,158.793
C08035=1023.768,-45.674,-94.152,166.779,48.163,158.793
C08036=1023.774,-45.424,-94.164,166.782,48.159,158.793
C08037=1023.779,-45.174,-94.175,166.786,48.156,158.793
C08038=1023.785,-44.924,-94.188,166.788,48.152,158.792
C08039=1023.792,-44.675,-94.200,166.792,48.149,158.792
C08040=1023.797,-44.426,-94.212,166.794,48.146,158.792
C08041=1023.803,-44.176,-94.224,166.797,48.142,158.792
C08042=1023.810,-43.925,-94.236,166.800,48.139,158.791
C08043=1023.815,-43.676,-94.248,166.803,48.136,158.791
C08044=1023.821,-43.427,-94.260,166.806,48.132,158.791
C08045=1023.827,-43.177,-94.272,166.809,48.129,158.791
C08046=1023.833,-42.928,-94.284,166.811,48.125,158.790
C08047=1023.839,-42.678,-94.296,166.814,48.122,158.790
C08048=1023.845,-42.428,-94.308,166.817,48.119,158.790
C08049=1023.851,-42.179,-94.320,166.820,48.115,158.790
C08050=1023.857,-41.929,-94.332,166.823,48.112,158.790
C08051=1023.863,-41.679,-94.345,166.826,48.109,158.790
C08052=1023.869,-41.430,-94.357,166.828,48.105,158.789
C08053=1023.875,-41.180,-94.369,166.831,48.102,158.789
C08054=1023.881,-40.931,-94.381,166.834,48.098,158.789
C08055=1023.887,-40.681,-94.394,166.838,48.095,158.789
C08056=1023.893,-40.432,-94.406,166.840,48.091,158.788
C08057=1023.899,-40.181,-94.417,166.844,48.088,158.788
C08058=1023.905,-39.931,-94.430,166.847,48.084,158.788
C08059=1023.911,-39.682,-94.442,166.849,48.081,158.788
C08060=1023.917,-39.433,-94.454,166.852,48.078,158.788
C08061=1023.923,-39.183,-94.466,166.855,48.074,158.787
C08062=1023.929,-38.933,-94.479,166.858,48.071,158.787
C08063=1023.935,-38.683,-94.491,166.861,48.067,158.787
C08064=1023.941,-38.434,-94.503,166.863,48.065,158.787
C08065=1023.947,-38.184,-94.516,166.866,48.061,158.786
C08066=1023.952,-37.934,-94.528,166.869,48.057,158.786
C08067=1023.959,-37.685,-94.541,166.872,48.054,158.786
C08068=1023.964,-37.436,-94.554,166.874,48.051,158.786
C08069=1023.970,-37.156,-94.567,166.878,48.047,158.786
C08070=1023.977,-36.877,-94.581,166.881,48.043,158.785
C08071=1023.984,-36.598,-94.595,166.884,48.039,158.785
C08072=1023.990,-36.318,-94.609,166.887,48.036,158.785
C08073=1023.997,-36.069,-94.622,166.890,48.032,158.785
C08074=1024.003,-35.819,-94.634,166.893,48.029,158.785
C08075=1024.009,-35.569,-94.647,166.896,48.026,158.784
C08076=1024.015,-35.319,-94.659,166.899,48.023,158.784
C08077=1024.020,-35.070,-94.672,166.902,48.019,158.784
C08078=1024.026,-34.820,-94.684,166.905,48.016,158.784
C08079=1024.032,-34.571,-94.697,166.908,48.013,158.784
C08080=1024.038,-34.321,-94.710,166.911,48.009,158.783
C08081=1024.044,-34.071,-94.723,166.913,48.006,158.783
C08082=1024.051,-33.821,-94.735,166.916,48.003,158.783
C08083=1024.056,-33.572,-94.747,166.919,47.999,158.783
C08084=1024.062,-33.323,-94.760,166.922,47.996,158.783
C08085=1024.068,-33.073,-94.773,166.924,47.993,158.782
C08086=1024.074,-32.823,-94.785,166.927,47.989,158.782
C08087=1024.080,-32.573,-94.798,166.930,47.986,158.782
C08088=1024.086,-32.324,-94.811,166.933,47.983,158.782
C08089=1024.092,-32.074,-94.823,166.935,47.979,158.781
C08090=1024.098,-31.824,-94.836,166.939,47.976,158.781
C08091=1024.103,-31.575,-94.848,166.941,47.972,158.781
C08092=1024.110,-31.326,-94.861,166.945,47.969,158.781
C08093=1024.116,-31.076,-94.873,166.948,47.966,158.781
C08094=1024.122,-30.826,-94.886,166.950,47.962,158.780
C08095=1024.128,-30.577,-94.899,166.953,47.959,158.780
C08096=1024.134,-30.327,-94.912,166.956,47.956,158.780
C08097=1024.140,-30.077,-94.924,166.959,47.952,158.780
C08098=1024.146,-29.828,-94.938,166.961,47.949,158.779
C08099=1024.152,-29.578,-94.950,166.964,47.945,158.779
C08100=1024.158,-29.328,-94.963,166.967,47.942,158.779
C08101=1024.164,-29.079,-94.976,166.970,47.939,158.779
C08102=1024.170,-28.829,-94.989,166.973,47.935,158.778
C08103=1024.177,-28.579,-95.001,166.975,47.932,158.778
C08104=1024.183,-28.330,-95.014,166.978,47.928,158.778
C08105=1024.189,-28.080,-95.026,166.981,47.925,158.778
C08106=1024.195,-27.830,-95.039,166.984,47.922,158.778
C08107=1024.200,-27.582,-95.052,166.987,47.918,158.777
C08108=1024.206,-27.332,-95.064,166.989,47.915,158.777
C08109=1024.212,-27.083,-95.078,166.992,47.911,158.777
C08110=1024.218,-26.833,-95.091,166.996,47.908,158.777
C08111=1024.224,-26.583,-95.104,166.998,47.905,158.776
C08112=1024.230,-26.333,-95.117,167.001,47.902,158.776
C08113=1024.236,-26.084,-95.130,167.004,47.898,158.776
C08114=1024.242,-25.834,-95.142,167.006,47.895,158.776
C08115=1024.248,-25.585,-95.156,167.009,47.892,158.776
C08116=1024.254,-25.335,-95.170,167.012,47.889,158.775
C08117=1024.259,-25.086,-95.182,167.015,47.885,158.775
C08118=1024.266,-24.836,-95.195,167.017,47.882,158.775
C08119=1024.272,-24.586,-95.208,167.021,47.879,158.775
C08120=1024.278,-24.337,-95.221,167.024,47.876,158.775
C08121=1024.283,-24.088,-95.235,167.026,47.872,158.774
C08122=1024.289,-23.838,-95.248,167.029,47.869,158.774
C08123=1024.295,-23.588,-95.261,167.032,47.866,158.774
C08124=1024.301,-23.338,-95.273,167.035,47.862,158.774
C08125=1024.308,-23.089,-95.287,167.037,47.859,158.773
C08126=1024.314,-22.839,-95.301,167.040,47.856,158.773
C08127=1024.320,-22.589,-95.314,167.043,47.852,158.773
C08128=1024.326,-22.340,-95.327,167.045,47.849,158.773
C08129=1024.332,-22.091,-95.340,167.048,47.846,158.773
C08130=1024.338,-21.841,-95.353,167.051,47.842,158.772
C08131=1024.343,-21.591,-95.366,167.053,47.840,158.772
C08132=1024.350,-21.342,-95.380,167.057,47.836,158.772
C08133=1024.356,-21.061,-95.394,167.059,47.833,158.772
C08134=1024.363,-20.781,-95.409,167.062,47.829,158.771
C08135=1024.370,-20.501,-95.424,167.066,47.825,158.771
C08136=1024.377,-20.221,-95.439,167.069,47.821,158.771
C08137=1024.383,-19.971,-95.452,167.072,47.818,158.771
C08138=1024.388,-19.721,-95.465,167.074,47.815,158.770
C08139=1024.394,-19.472,-95.478,167.078,47.812,158.770
C08140=1024.401,-19.223,-95.492,167.081,47.808,158.770
C08141=1024.407,-18.973,-95.505,167.083,47.805,158.770
C08142=1024.413,-18.723,-95.518,167.086,47.802,158.769
C08143=1024.419,-18.473,-95.532,167.089,47.798,158.769
C08144=1024.425,-18.224,-95.545,167.092,47.795,158.769
C08145=1024.431,-17.975,-95.558,167.094,47.791,158.769
C08146=1024.437,-17.725,-95.571,167.097,47.788,158.768
C08147=1024.443,-17.475,-95.585,167.100,47.785,158.768
C08148=1024.449,-17.225,-95.598,167.102,47.781,158.768
C08149=1024.456,-16.976,-95.612,167.105,47.778,158.768
C08150=1024.462,-16.727,-95.625,167.108,47.774,158.767
C08151=1024.468,-16.477,-95.637,167.111,47.771,158.767
C08152=1024.473,-16.227,-95.651,167.113,47.768,158.767
C08153=1024.480,-15.977,-95.665,167.116,47.764,158.767
C08154=1024.486,-15.728,-95.678,167.119,47.761,158.767
C08155=1024.492,-15.478,-95.692,167.121,47.758,158.766
C08156=1024.498,-15.229,-95.705,167.125,47.754,158.766
C08157=1024.503,-14.980,-95.719,167.128,47.751,158.766
C08158=1024.510,-14.730,-95.733,167.130,47.748,158.766
C08159=1024.516,-14.480,-95.747,167.133,47.745,158.765
C08160=1024.522,-14.231,-95.760,167.135,47.742,158.765
C08161=1024.527,-13.981,-95.774,167.138,47.739,158.765
C08162=1024.534,-13.732,-95.787,167.141,47.735,158.765
C08163=1024.540,-13.482,-95.801,167.143,47.732,158.764
C08164=1024.546,-13.232,-95.815,167.146,47.729,158.764
C08165=1024.551,-12.983,-95.828,167.150,47.726,158.764
C08166=1024.558,-12.734,-95.842,167.151,47.722,158.764
C08167=1024.563,-12.484,-95.856,167.155,47.719,158.764
C08168=1024.570,-12.234,-95.869,167.158,47.716,158.763
C08169=1024.575,-11.984,-95.883,167.160,47.713,158.763
C08170=1024.582,-11.735,-95.896,167.163,47.709,158.763
C08171=1024.587,-11.486,-95.910,167.166,47.706,158.763
C08172=1024.594,-11.236,-95.924,167.168,47.703,158.762
C08173=1024.599,-10.986,-95.938,167.171,47.699,158.762
C08174=1024.606,-10.737,-95.951,167.173,47.696,158.762
C08175=1024.611,-10.487,-95.965,167.176,47.693,158.762
C08176=1024.618,-10.238,-95.979,167.179,47.689,158.761
C08177=1024.624,-9.988,-95.993,167.181,47.686,158.761
C08178=1024.630,-9.739,-96.006,167.185,47.683,158.761
C08179=1024.636,-9.489,-96.021,167.188,47.679,158.761
C08180=1024.642,-9.239,-96.034,167.190,47.677,158.761
C08181=1024.648,-8.990,-96.048,167.193,47.673,158.760
C08182=1024.654,-8.741,-96.061,167.196,47.670,158.760
C08183=1024.660,-8.490,-96.075,167.198,47.667,158.760
C08184=1024.666,-8.242,-96.089,167.201,47.663,158.759
C08185=1024.672,-7.992,-96.103,167.204,47.660,158.759
C08186=1024.679,-7.742,-96.117,167.206,47.657,158.759
C08187=1024.684,-7.493,-96.131,167.209,47.653,158.759
C08188=1024.690,-7.243,-96.144,167.211,47.650,158.759
C08189=1024.697,-6.994,-96.159,167.214,47.647,158.758
C08190=1024.703,-6.744,-96.172,167.217,47.643,158.758
C08191=1024.708,-6.495,-96.186,167.219,47.640,158.758
C08192=1024.715,-6.245,-96.200,167.222,47.637,158.758
C08193=1024.721,-5.995,-96.213,167.226,47.633,158.757
C08194=1024.728,-5.746,-96.228,167.228,47.631,158.757
C08195=1024.733,-5.496,-96.242,167.231,47.627,158.757
C08196=1024.740,-5.247,-96.255,167.234,47.624,158.757
C08197=1024.746,-4.965,-96.272,167.237,47.620,158.756
C08198=1024.754,-4.683,-96.287,167.240,47.616,158.756
C08199=1024.760,-4.401,-96.302,167.242,47.612,158.756
C08200=1024.768,-4.119,-96.318,167.245,47.608,158.755
C08201=1024.773,-3.869,-96.332,167.249,47.605,158.755
C08202=1024.780,-3.620,-96.347,167.251,47.602,158.755
C08203=1024.785,-3.370,-96.361,167.254,47.599,158.755
C08204=1024.791,-3.120,-96.375,167.256,47.596,158.754
C08205=1024.797,-2.871,-96.390,167.259,47.592,158.754
C08206=1024.802,-2.621,-96.403,167.262,47.589,158.754
C08207=1024.809,-2.372,-96.418,167.264,47.586,158.754
C08208=1024.815,-2.122,-96.432,167.268,47.583,158.754
C08209=1024.821,-1.873,-96.446,167.269,47.580,158.753
C08210=1024.827,-1.623,-96.461,167.273,47.577,158.753
C08211=1024.833,-1.374,-96.475,167.275,47.574,158.753
C08212=1024.839,-1.124,-96.489,167.278,47.571,158.753
C08213=1024.844,-0.875,-96.504,167.280,47.567,158.752
C08214=1024.851,-0.625,-96.518,167.283,47.564,158.752
C08215=1024.856,-0.376,-96.533,167.286,47.561,158.752
C08216=1024.863,-0.127,-96.546,167.288,47.558,158.752
C08217=1024.869,0.123,-96.561,167.291,47.554,158.751
C08218=1024.874,0.373,-96.575,167.293,47.551,158.751
///RCONF 1,0,0,0,0,0,0,0,0,0,0,0,0,0,0,0,0,0,0,0,0,0,0,0
C08219=1024.881,0.622,-96.590,167.297,47.548,158.751
C08220=1024.886,0.872,-96.604,167.299,47.545,158.751
C08221=1024.893,1.122,-96.619,167.302,47.542,158.751
C08222=1024.898,1.371,-96.632,167.304,47.539,158.750
C08223=1024.905,1.621,-96.647,167.307,47.536,158.750
C08224=1024.910,1.870,-96.662,167.310,47.532,158.750
C08225=1024.917,2.119,-96.675,167.312,47.529,158.750
C08226=1024.923,2.369,-96.690,167.315,47.526,158.749
C08227=1024.928,2.618,-96.704,167.317,47.522,158.749
C08228=1024.935,2.868,-96.719,167.320,47.519,158.749
C08229=1024.941,3.117,-96.734,167.323,47.516,158.749
C08230=1024.947,3.367,-96.748,167.326,47.513,158.748
C08231=1024.952,3.616,-96.762,167.328,47.510,158.748
C08232=1024.958,3.866,-96.777,167.331,47.506,158.748
C08233=1024.964,4.115,-96.791,167.334,47.503,158.748
C08234=1024.971,4.365,-96.806,167.336,47.500,158.747
C08235=1024.977,4.615,-96.820,167.339,47.497,158.747
C08236=1024.983,4.864,-96.834,167.341,47.494,158.747
C08237=1024.990,5.114,-96.849,167.344,47.490,158.747
C08238=1024.995,5.363,-96.863,167.346,47.487,158.746
C08239=1025.001,5.613,-96.878,167.350,47.484,158.746
C08240=1025.007,5.862,-96.893,167.352,47.480,158.746
C08241=1025.013,6.112,-96.907,167.355,47.477,158.746
C08242=1025.019,6.361,-96.921,167.358,47.474,158.745
C08243=1025.026,6.611,-96.936,167.360,47.471,158.745
C08244=1025.031,6.860,-96.951,167.363,47.468,158.745
C08245=1025.037,7.110,-96.965,167.365,47.464,158.744
C08246=1025.044,7.360,-96.980,167.368,47.461,158.744
C08247=1025.050,7.608,-96.994,167.371,47.458,158.744
C08248=1025.057,7.858,-97.009,167.373,47.454,158.744
C08249=1025.064,8.181,-97.028,167.377,47.450,158.743
C08250=1025.072,8.503,-97.047,167.380,47.446,158.743
C08251=1025.080,8.826,-97.066,167.383,47.442,158.743
C08252=1025.088,9.148,-97.085,167.387,47.438,158.742
C08253=1025.094,9.398,-97.098,167.389,47.434,158.742
C08254=1025.100,9.647,-97.113,167.392,47.431,158.742
C08255=1025.106,9.897,-97.128,167.394,47.427,158.741
C08256=1025.112,10.146,-97.143,167.398,47.424,158.741
C08257=1025.118,10.376,-97.156,167.400,47.421,158.741
C08258=1025.124,10.607,-97.170,167.402,47.418,158.741
C08259=1025.130,10.837,-97.183,167.405,47.415,158.741
C08260=1025.135,11.067,-97.197,167.407,47.412,158.740
C08261=1025.141,11.297,-97.210,167.409,47.409,158.740
C08262=1025.146,11.527,-97.224,167.412,47.406,158.740
C08263=1025.152,11.757,-97.237,167.415,47.403,158.740
C08264=1025.158,11.988,-97.251,167.416,47.400,158.739
C08265=1025.164,12.237,-97.266,167.420,47.396,158.739
C08266=1025.170,12.486,-97.281,167.421,47.393,158.739
C08267=1025.177,12.736,-97.296,167.425,47.390,158.738
C08268=1025.182,12.985,-97.310,167.428,47.386,158.738
C08269=1025.188,13.235,-97.324,167.430,47.383,158.738
C08270=1025.195,13.485,-97.339,167.433,47.380,158.738
C08271=1025.201,13.734,-97.354,167.435,47.377,158.737
C08272=1025.207,13.984,-97.369,167.438,47.373,158.737
C08273=1025.213,14.233,-97.384,167.440,47.371,158.737
C08274=1025.220,14.483,-97.399,167.443,47.367,158.737
C08275=1025.226,14.732,-97.413,167.445,47.364,158.736
C08276=1025.231,14.982,-97.429,167.449,47.361,158.736
C08277=1025.238,15.231,-97.444,167.450,47.357,158.736
C08278=1025.243,15.480,-97.459,167.454,47.354,158.736
C08279=1025.250,15.729,-97.474,167.456,47.351,158.735
C08280=1025.256,15.979,-97.490,167.459,47.348,158.735
C08281=1025.262,16.228,-97.504,167.461,47.345,158.735
C08282=1025.268,16.478,-97.519,167.464,47.342,158.735
C08283=1025.274,16.728,-97.534,167.466,47.338,158.734
C08284=1025.281,16.977,-97.549,167.469,47.335,158.734
C08285=1025.286,17.227,-97.564,167.471,47.331,158.734
C08286=1025.292,17.476,-97.579,167.474,47.328,158.733
C08287=1025.298,17.726,-97.594,167.476,47.326,158.733
C08288=1025.305,17.976,-97.609,167.479,47.322,158.733
C08289=1025.311,18.224,-97.624,167.483,47.319,158.733
C08290=1025.317,18.474,-97.640,167.485,47.316,158.732
C08291=1025.323,18.723,-97.655,167.488,47.312,158.732
C08292=1025.329,18.973,-97.670,167.490,47.309,158.732
C08293=1025.335,19.222,-97.684,167.493,47.305,158.732
C08294=1025.341,19.472,-97.700,167.495,47.303,158.731
C08295=1025.347,19.721,-97.716,167.498,47.299,158.731
C08296=1025.354,19.971,-97.731,167.500,47.296,158.731
C08297=1025.359,20.220,-97.746,167.503,47.293,158.731
C08298=1025.365,20.470,-97.761,167.505,47.290,158.730
C08299=1025.371,20.720,-97.776,167.507,47.286,158.730
C08300=1025.378,20.969,-97.792,167.510,47.283,158.730
C08301=1025.384,21.218,-97.807,167.513,47.281,158.729
C08302=1025.389,21.468,-97.822,167.516,47.277,158.729
C08303=1025.396,21.717,-97.838,167.518,47.274,158.729
C08304=1025.402,21.966,-97.853,167.521,47.271,158.729
C08305=1025.408,22.216,-97.868,167.523,47.267,158.728
C08306=1025.414,22.466,-97.883,167.526,47.264,158.728
C08307=1025.420,22.714,-97.898,167.528,47.261,158.728
C08308=1025.426,22.964,-97.914,167.531,47.258,158.728
C08309=1025.432,23.214,-97.929,167.533,47.255,158.727
C08310=1025.438,23.463,-97.945,167.536,47.252,158.727
C08311=1025.445,23.713,-97.960,167.538,47.248,158.727
C08312=1025.451,23.963,-97.975,167.542,47.245,158.727
C08313=1025.456,24.211,-97.991,167.543,47.241,158.726
C08314=1025.463,24.461,-98.006,167.547,47.238,158.726
C08315=1025.468,24.711,-98.021,167.549,47.236,158.726
C08316=1025.475,24.960,-98.037,167.552,47.232,158.725
C08317=1025.481,25.210,-98.052,167.554,47.229,158.725
C08318=1025.487,25.459,-98.068,167.557,47.225,158.725
C08319=1025.494,25.709,-98.083,167.559,47.222,158.725
C08320=1025.500,25.957,-98.098,167.562,47.219,158.724
C08321=1025.506,26.207,-98.114,167.564,47.216,158.724
C08322=1025.512,26.456,-98.129,167.567,47.213,158.724
C08323=1025.518,26.706,-98.145,167.569,47.209,158.723
C08324=1025.524,26.955,-98.160,167.572,47.206,158.723
C08325=1025.531,27.241,-98.179,167.575,47.202,158.723
C08326=1025.538,27.526,-98.196,167.578,47.199,158.723
C08327=1025.545,27.811,-98.214,167.581,47.195,158.722
C08328=1025.552,28.097,-98.231,167.584,47.192,158.722
C08329=1025.558,28.346,-98.247,167.586,47.188,158.722
C08330=1025.565,28.595,-98.263,167.588,47.185,158.721
C08331=1025.570,28.845,-98.279,167.592,47.182,158.721
C08332=1025.576,29.094,-98.294,167.594,47.179,158.721
C08333=1025.582,29.344,-98.309,167.597,47.176,158.721
C08334=1025.588,29.593,-98.326,167.599,47.173,158.720
C08335=1025.594,29.843,-98.341,167.602,47.169,158.720
C08336=1025.600,30.092,-98.357,167.604,47.166,158.720
C08337=1025.606,30.341,-98.373,167.607,47.163,158.720
C08338=1025.613,30.591,-98.388,167.609,47.160,158.719
C08339=1025.619,30.840,-98.404,167.611,47.157,158.719
C08340=1025.624,31.090,-98.420,167.615,47.154,158.719
C08341=1025.631,31.339,-98.435,167.616,47.150,158.718
C08342=1025.637,31.589,-98.452,167.620,47.147,158.718
C08343=1025.642,31.839,-98.467,167.622,47.144,158.718
C08344=1025.649,32.088,-98.483,167.625,47.141,158.718
C08345=1025.655,32.337,-98.499,167.627,47.138,158.717
C08346=1025.662,32.587,-98.514,167.630,47.135,158.717
C08347=1025.667,32.835,-98.530,167.632,47.131,158.717
C08348=1025.673,33.085,-98.546,167.634,47.128,158.716
C08349=1025.679,33.334,-98.561,167.637,47.125,158.716
C08350=1025.685,33.584,-98.577,167.639,47.122,158.716
C08351=1025.691,33.833,-98.594,167.643,47.119,158.716
C08352=1025.697,34.083,-98.609,167.644,47.115,158.715
C08353=1025.703,34.332,-98.625,167.648,47.112,158.715
C08354=1025.709,34.581,-98.641,167.650,47.109,158.715
C08355=1025.716,34.831,-98.656,167.653,47.105,158.715
C08356=1025.722,35.080,-98.672,167.655,47.103,158.714
C08357=1025.728,35.329,-98.688,167.658,47.099,158.714
C08358=1025.734,35.579,-98.704,167.660,47.096,158.714
C08359=1025.740,35.829,-98.720,167.663,47.092,158.713
C08360=1025.747,36.078,-98.736,167.665,47.089,158.713
C08361=1025.753,36.328,-98.752,167.667,47.087,158.713
C08362=1025.759,36.577,-98.768,167.670,47.083,158.712
C08363=1025.766,36.827,-98.783,167.673,47.080,158.712
C08364=1025.772,37.076,-98.800,167.675,47.076,158.712
C08365=1025.777,37.325,-98.816,167.678,47.073,158.712
C08366=1025.783,37.575,-98.832,167.681,47.070,158.711
C08367=1025.789,37.824,-98.848,167.683,47.067,158.711
C08368=1025.795,38.074,-98.865,167.685,47.064,158.711
C08369=1025.801,38.323,-98.880,167.688,47.061,158.711
C08370=1025.808,38.573,-98.896,167.690,47.058,158.710
C08371=1025.814,38.822,-98.912,167.693,47.054,158.710
C08372=1025.820,39.071,-98.928,167.695,47.052,158.710
C08373=1025.826,39.321,-98.945,167.699,47.049,158.710
C08374=1025.831,39.570,-98.961,167.701,47.045,158.709
C08375=1025.837,39.819,-98.977,167.703,47.042,158.709
C08376=1025.843,40.069,-98.993,167.706,47.039,158.709
C08377=1025.849,40.318,-99.010,167.708,47.036,158.708
C08378=1025.855,40.567,-99.026,167.711,47.033,158.708
C08379=1025.862,40.816,-99.042,167.713,47.029,158.708
C08380=1025.869,41.066,-99.058,167.715,47.026,158.707
C08381=1025.874,41.316,-99.074,167.718,47.023,158.707
C08382=1025.880,41.565,-99.091,167.720,47.020,158.707
C08383=1025.886,41.814,-99.107,167.724,47.017,158.707
C08384=1025.892,42.064,-99.123,167.726,47.014,158.706
C08385=1025.898,42.313,-99.139,167.729,47.010,158.706
C08386=1025.904,42.562,-99.156,167.731,47.007,158.706
C08387=1025.910,42.812,-99.172,167.733,47.004,158.706
C08388=1025.916,43.061,-99.188,167.736,47.001,158.705
C08389=1025.923,43.347,-99.207,167.739,46.998,158.705
C08390=1025.930,43.632,-99.225,167.741,46.994,158.705
C08391=1025.936,43.917,-99.244,167.744,46.990,158.704
C08392=1025.943,44.202,-99.263,167.747,46.987,158.704
C08393=1025.949,44.452,-99.280,167.749,46.984,158.704
C08394=1025.956,44.702,-99.296,167.752,46.981,158.704
C08395=1025.962,44.950,-99.313,167.755,46.978,158.703
C08396=1025.967,45.200,-99.330,167.758,46.975,158.703
C08397=1025.973,45.450,-99.346,167.760,46.971,158.703
C08398=1025.979,45.699,-99.363,167.762,46.969,158.702
C08399=1025.985,45.948,-99.379,167.765,46.966,158.702
C08400=1025.991,46.198,-99.395,167.767,46.963,158.702
C08401=1025.997,46.446,-99.412,167.769,46.959,158.702
C08402=1026.003,46.697,-99.429,167.772,46.956,158.701
C08403=1026.009,46.946,-99.446,167.775,46.953,158.701
C08404=1026.015,47.195,-99.462,167.777,46.951,158.701
C08405=1026.021,47.444,-99.479,167.780,46.947,158.701
C08406=1026.027,47.693,-99.495,167.782,46.944,158.700
C08407=1026.032,47.943,-99.512,167.785,46.941,158.700
C08408=1026.039,48.193,-99.528,167.787,46.937,158.700
C08409=1026.045,48.442,-99.545,167.789,46.935,158.699
C08410=1026.051,48.691,-99.562,167.792,46.932,158.699
C08411=1026.057,48.941,-99.578,167.794,46.928,158.699
C08412=1026.063,49.190,-99.594,167.797,46.925,158.699
C08413=1026.069,49.439,-99.612,167.800,46.922,158.698
C08414=1026.075,49.689,-99.628,167.802,46.919,158.698
C08415=1026.081,49.938,-99.645,167.805,46.916,158.698
C08416=1026.087,50.188,-99.661,167.807,46.913,158.697
C08417=1026.093,50.436,-99.678,167.809,46.910,158.697
C08418=1026.099,50.687,-99.695,167.812,46.906,158.697
C08419=1026.105,50.936,-99.711,167.814,46.904,158.697
C08420=1026.111,51.185,-99.728,167.818,46.901,158.696
C08421=1026.117,51.434,-99.745,167.820,46.897,158.696
C08422=1026.123,51.684,-99.761,167.822,46.894,158.696
C08423=1026.129,51.933,-99.779,167.825,46.891,158.695
C08424=1026.135,52.183,-99.795,167.827,46.888,158.695
C08425=1026.141,52.432,-99.811,167.830,46.885,158.695
C08426=1026.147,52.681,-99.828,167.832,46.881,158.695
C08427=1026.154,52.931,-99.845,167.834,46.878,158.694
C08428=1026.160,53.180,-99.862,167.837,46.875,158.694
C08429=1026.165,53.429,-99.879,167.839,46.872,158.694
C08430=1026.172,53.679,-99.895,167.843,46.869,158.694
C08431=1026.178,53.928,-99.912,167.845,46.865,158.693
C08432=1026.184,54.177,-99.929,167.847,46.863,158.693
C08433=1026.190,54.426,-99.946,167.850,46.859,158.693
C08434=1026.196,54.676,-99.963,167.852,46.856,158.692
C08435=1026.202,54.926,-99.979,167.855,46.853,158.692
C08436=1026.209,55.174,-99.996,167.857,46.849,158.692
C08437=1026.215,55.425,-100.013,167.859,46.847,158.691
C08438=1026.221,55.674,-100.030,167.862,46.844,158.691
C08439=1026.227,55.923,-100.046,167.864,46.840,158.691
C08440=1026.233,56.172,-100.064,167.868,46.837,158.691
C08441=1026.239,56.422,-100.080,167.869,46.834,158.690
C08442=1026.245,56.671,-100.098,167.872,46.831,158.690
C08443=1026.251,56.920,-100.114,167.875,46.828,158.690
C08444=1026.258,57.169,-100.131,167.877,46.824,158.689
C08445=1026.264,57.419,-100.147,167.880,46.821,158.689
C08446=1026.270,57.668,-100.165,167.882,46.818,158.689
C08447=1026.276,57.918,-100.182,167.885,46.815,158.688
C08448=1026.282,58.167,-100.199,167.887,46.811,158.688
C08449=1026.289,58.417,-100.215,167.889,46.808,158.688
C08450=1026.295,58.665,-100.232,167.892,46.805,158.687
C08451=1026.300,58.915,-100.249,167.894,46.802,158.687
C08452=1026.307,59.165,-100.266,167.897,46.798,158.687
C08453=1026.314,59.449,-100.285,167.900,46.794,158.686
C08454=1026.321,59.734,-100.304,167.903,46.791,158.686
C08455=1026.328,60.019,-100.323,167.905,46.787,158.686
C08456=1026.335,60.304,-100.344,167.908,46.784,158.686
C08457=1026.341,60.554,-100.360,167.911,46.781,158.685
C08458=1026.348,60.803,-100.377,167.914,46.778,158.685
C08459=1026.354,61.052,-100.394,167.916,46.774,158.685
C08460=1026.360,61.302,-100.411,167.919,46.771,158.684
C08461=1026.366,61.551,-100.428,167.922,46.768,158.684
C08462=1026.373,61.800,-100.445,167.924,46.764,158.684
C08463=1026.379,62.049,-100.462,167.927,46.761,158.683
C08464=1026.385,62.300,-100.479,167.929,46.758,158.683
C08465=1026.391,62.548,-100.496,167.931,46.755,158.683
C08466=1026.397,62.797,-100.513,167.934,46.751,158.682
C08467=1026.404,63.047,-100.530,167.936,46.748,158.682
C08468=1026.409,63.296,-100.547,167.939,46.745,158.682
C08469=1026.416,63.546,-100.565,167.941,46.742,158.681
C08470=1026.421,63.795,-100.582,167.944,46.739,158.681
C08471=1026.428,64.045,-100.599,167.946,46.735,158.681
C08472=1026.434,64.294,-100.616,167.949,46.732,158.681
C08473=1026.440,64.542,-100.633,167.952,46.729,158.680
C08474=1026.446,64.793,-100.651,167.954,46.726,158.680
C08475=1026.452,65.041,-100.668,167.956,46.723,158.680
C08476=1026.458,65.291,-100.686,167.959,46.719,158.679
C08477=1026.464,65.540,-100.703,167.961,46.717,158.679
C08478=1026.470,65.790,-100.720,167.964,46.714,158.679
C08479=1026.476,66.039,-100.737,167.966,46.710,158.678
C08480=1026.482,66.288,-100.754,167.968,46.707,158.678
C08481=1026.488,66.538,-100.772,167.972,46.704,158.678
C08482=1026.494,66.787,-100.789,167.974,46.701,158.678
C08483=1026.500,67.036,-100.807,167.977,46.698,158.677
C08484=1026.507,67.285,-100.824,167.979,46.694,158.677
C08485=1026.513,67.535,-100.842,167.981,46.692,158.677
C08486=1026.519,67.784,-100.858,167.984,46.689,158.676
C08487=1026.525,68.034,-100.876,167.986,46.685,158.676
C08488=1026.530,68.283,-100.894,167.988,46.682,158.676
C08489=1026.537,68.532,-100.911,167.991,46.679,158.675
C08490=1026.543,68.781,-100.929,167.993,46.676,158.675
C08491=1026.549,69.031,-100.947,167.997,46.673,158.675
C08492=1026.555,69.280,-100.964,167.999,46.669,158.675
C08493=1026.561,69.530,-100.982,168.001,46.667,158.674
C08494=1026.567,69.779,-100.999,168.004,46.664,158.674
C08495=1026.574,70.028,-101.016,168.006,46.660,158.674
C08496=1026.579,70.277,-101.034,168.008,46.657,158.673
C08497=1026.585,70.527,-101.052,168.011,46.654,158.673
C08498=1026.591,70.776,-101.070,168.013,46.651,158.673
C08499=1026.598,71.025,-101.087,168.017,46.648,158.673
C08500=1026.603,71.274,-101.104,168.019,46.645,158.672
C08501=1026.609,71.524,-101.122,168.021,46.642,158.672
C08502=1026.615,71.773,-101.140,168.024,46.639,158.672
C08503=1026.622,72.023,-101.157,168.026,46.636,158.671
C08504=1026.627,72.272,-101.175,168.028,46.632,158.671
C08505=1026.633,72.521,-101.193,168.031,46.629,158.671
C08506=1026.639,72.770,-101.210,168.034,46.627,158.671
C08507=1026.646,73.020,-101.228,168.036,46.623,158.670
C08508=1026.651,73.269,-101.245,168.039,46.620,158.670
C08509=1026.657,73.519,-101.263,168.041,46.617,158.670
C08510=1026.664,73.768,-101.282,168.044,46.614,158.669
C08511=1026.669,74.017,-101.299,168.046,46.611,158.669
C08512=1026.676,74.266,-101.317,168.048,46.608,158.669
C08513=1026.682,74.515,-101.334,168.051,46.604,158.668
C08514=1026.688,74.765,-101.352,168.053,46.602,158.668
C08515=1026.693,75.014,-101.370,168.056,46.598,158.668
C08516=1026.700,75.263,-101.387,168.059,46.595,158.668
C08517=1026.707,75.548,-101.407,168.062,46.591,158.667
C08518=1026.714,75.833,-101.428,168.064,46.588,158.667
C08519=1026.721,76.118,-101.448,168.067,46.584,158.666
C08520=1026.727,76.403,-101.469,168.069,46.581,158.666
C08521=1026.734,76.652,-101.487,168.073,46.577,158.666
C08522=1026.739,76.901,-101.504,168.075,46.575,158.666
C08523=1026.745,77.150,-101.523,168.078,46.571,158.665
C08524=1026.752,77.400,-101.540,168.080,46.568,158.665
C08525=1026.758,77.649,-101.558,168.082,46.565,158.665
C08526=1026.764,77.899,-101.576,168.085,46.562,158.664
C08527=1026.770,78.148,-101.594,168.087,46.559,158.664
C08528=1026.776,78.397,-101.612,168.090,46.556,158.664
C08529=1026.782,78.647,-101.630,168.093,46.553,158.664
C08530=1026.788,78.895,-101.648,168.095,46.550,158.663
C08531=1026.793,79.145,-101.667,168.097,46.547,158.663
C08532=1026.799,79.395,-101.685,168.100,46.544,158.663
C08533=1026.805,79.643,-101.703,168.102,46.541,158.662
C08534=1026.811,79.893,-101.721,168.104,46.538,158.662
C08535=1026.817,80.142,-101.738,168.108,46.535,158.662
C08536=1026.823,80.391,-101.757,168.110,46.532,158.662
C08537=1026.829,80.641,-101.775,168.113,46.528,158.661
C08538=1026.835,80.889,-101.793,168.115,46.526,158.661
C08539=1026.841,81.139,-101.811,168.117,46.523,158.661
C08540=1026.847,81.389,-101.829,168.120,46.519,158.660
C08541=1026.853,81.637,-101.847,168.122,46.516,158.660
C08542=1026.859,81.887,-101.865,168.125,46.514,158.660
C08543=1026.866,82.137,-101.883,168.128,46.510,158.659
C08544=1026.871,82.385,-101.902,168.130,46.507,158.659
C08545=1026.877,82.635,-101.919,168.132,46.504,158.659
C08546=1026.884,82.884,-101.938,168.135,46.501,158.659
C08547=1026.889,83.133,-101.956,168.137,46.498,158.658
C08548=1026.895,83.382,-101.975,168.140,46.495,158.658
C08549=1026.901,83.632,-101.993,168.142,46.491,158.658
C08550=1026.907,83.881,-102.011,168.145,46.489,158.657
C08551=1026.913,84.130,-102.029,168.148,46.486,158.657
C08552=1026.919,84.380,-102.047,168.150,46.482,158.657
C08553=1026.925,84.628,-102.065,168.152,46.479,158.656
C08554=1026.931,84.878,-102.083,168.155,46.476,158.656
C08555=1026.938,85.127,-102.102,168.157,46.473,158.656
C08556=1026.944,85.377,-102.120,168.160,46.470,158.656
C08557=1026.950,85.625,-102.138,168.163,46.467,158.655
C08558=1026.956,85.875,-102.156,168.165,46.464,158.655
C08559=1026.962,86.124,-102.175,168.168,46.461,158.655
C08560=1026.968,86.374,-102.193,168.170,46.457,158.654
C08561=1026.974,86.622,-102.211,168.173,46.454,158.654
C08562=1026.980,86.872,-102.230,168.175,46.452,158.654
C08563=1026.986,87.122,-102.248,168.177,46.448,158.653
C08564=1026.992,87.370,-102.266,168.180,46.445,158.653
C08565=1026.998,87.620,-102.284,168.183,46.442,158.653
C08566=1027.004,87.869,-102.303,168.186,46.439,158.653
C08567=1027.010,88.119,-102.321,168.188,46.436,158.652
C08568=1027.017,88.368,-102.339,168.191,46.432,158.652
C08569=1027.022,88.617,-102.357,168.193,46.430,158.652
C08570=1027.029,88.866,-102.376,168.195,46.427,158.651
C08571=1027.035,89.115,-102.394,168.198,46.423,158.651
C08572=1027.041,89.365,-102.412,168.200,46.420,158.651
C08573=1027.047,89.614,-102.432,168.203,46.417,158.650
C08574=1027.053,89.863,-102.450,168.205,46.414,158.650
C08575=1027.059,90.112,-102.468,168.208,46.411,158.650
C08576=1027.065,90.362,-102.487,168.211,46.408,158.650
C08577=1027.071,90.611,-102.506,168.213,46.405,158.649
C08578=1027.077,90.860,-102.523,168.215,46.402,158.649
C08579=1027.082,91.109,-102.542,168.218,46.399,158.649
C08580=1027.089,91.359,-102.561,168.221,46.396,158.649
C08581=1027.096,91.644,-102.583,168.224,46.393,158.648
C08582=1027.102,91.928,-102.603,168.227,46.389,158.648
C08583=1027.109,92.213,-102.625,168.229,46.385,158.647
C08584=1027.116,92.497,-102.646,168.232,46.382,158.647
C08585=1027.121,92.747,-102.665,168.235,46.379,158.647
C08586=1027.128,92.996,-102.684,168.237,46.376,158.647
C08587=1027.134,93.246,-102.703,168.240,46.373,158.646
C08588=1027.139,93.494,-102.721,168.242,46.370,158.646
C08589=1027.146,93.743,-102.740,168.244,46.367,158.646
C08590=1027.151,93.993,-102.759,168.248,46.364,158.645
C08591=1027.158,94.242,-102.777,168.250,46.361,158.645
C08592=1027.164,94.492,-102.796,168.253,46.357,158.645
C08593=1027.170,94.741,-102.815,168.255,46.355,158.645
C08594=1027.176,94.989,-102.833,168.257,46.352,158.644
C08595=1027.181,95.239,-102.852,168.260,46.348,158.644
C08596=1027.188,95.488,-102.871,168.262,46.346,158.644
C08597=1027.194,95.737,-102.890,168.266,46.343,158.643
C08598=1027.199,95.987,-102.908,168.268,46.339,158.643
C08599=1027.206,96.236,-102.927,168.270,46.336,158.643
C08600=1027.212,96.486,-102.946,168.273,46.333,158.643
C08601=1027.217,96.734,-102.964,168.275,46.330,158.642
C08602=1027.224,96.983,-102.983,168.278,46.327,158.642
C08603=1027.229,97.233,-103.002,168.280,46.324,158.642
C08604=1027.236,97.482,-103.021,168.282,46.321,158.641
C08605=1027.242,97.731,-103.040,168.286,46.318,158.641
C08606=1027.248,97.980,-103.059,168.288,46.315,158.641
C08607=1027.254,98.229,-103.077,168.291,46.311,158.640
C08608=1027.260,98.479,-103.097,168.293,46.309,158.640
C08609=1027.267,98.728,-103.115,168.295,46.306,158.640
C08610=1027.271,98.977,-103.133,168.298,46.302,158.639
C08611=1027.278,99.227,-103.152,168.301,46.300,158.639
C08612=1027.284,99.476,-103.171,168.303,46.296,158.639
C08613=1027.290,99.725,-103.190,168.306,46.293,158.638
C08614=1027.296,99.974,-103.209,168.309,46.290,158.638
C08615=1027.302,100.223,-103.229,168.311,46.287,158.638
C08616=1027.308,100.472,-103.248,168.313,46.284,158.638
C08617=1027.314,100.722,-103.267,168.316,46.281,158.637
C08618=1027.320,100.971,-103.286,168.319,46.278,158.637
C08619=1027.326,101.220,-103.305,168.321,46.276,158.637
C08620=1027.331,101.470,-103.324,168.324,46.273,158.637
C08621=1027.338,101.719,-103.343,168.326,46.269,158.636
C08622=1027.344,101.968,-103.362,168.329,46.266,158.636
C08623=1027.349,102.218,-103.381,168.332,46.263,158.636
C08624=1027.355,102.466,-103.400,168.334,46.261,158.635
C08625=1027.361,102.715,-103.420,168.337,46.257,158.635
C08626=1027.367,102.965,-103.439,168.339,46.254,158.635
C08627=1027.373,103.214,-103.457,168.342,46.251,158.635
C08628=1027.379,103.463,-103.477,168.344,46.249,158.634
C08629=1027.385,103.712,-103.496,168.346,46.245,158.634
C08630=1027.391,103.961,-103.516,168.350,46.242,158.634
C08631=1027.397,104.210,-103.535,168.352,46.239,158.633
C08632=1027.403,104.460,-103.554,168.355,46.236,158.633
C08633=1027.408,104.709,-103.573,168.357,46.233,158.633
C08634=1027.415,104.958,-103.592,168.359,46.230,158.632
C08635=1027.421,105.207,-103.612,168.363,46.227,158.632
C08636=1027.426,105.457,-103.631,168.365,46.225,158.632
C08637=1027.433,105.706,-103.650,168.368,46.221,158.632
C08638=1027.439,105.955,-103.669,168.370,46.218,158.631
C08639=1027.445,106.204,-103.689,168.372,46.215,158.631
C08640=1027.450,106.453,-103.708,168.375,46.212,158.631
C08641=1027.457,106.703,-103.727,168.377,46.209,158.630
C08642=1027.463,106.951,-103.747,168.381,46.206,158.630
C08643=1027.468,107.201,-103.766,168.383,46.203,158.630
C08644=1027.475,107.450,-103.784,168.386,46.200,158.630
C08645=1027.482,107.735,-103.806,168.389,46.196,158.629
C08646=1027.489,108.019,-103.829,168.391,46.193,158.629
C08647=1027.496,108.304,-103.851,168.394,46.190,158.629
C08648=1027.502,108.589,-103.873,168.397,46.186,158.628
C08649=1027.508,108.839,-103.892,168.400,46.183,158.628
C08650=1027.515,109.087,-103.912,168.403,46.180,158.628
C08651=1027.521,109.337,-103.931,168.405,46.177,158.627
C08652=1027.526,109.586,-103.950,168.408,46.174,158.627
C08653=1027.532,109.835,-103.970,168.411,46.171,158.627
C08654=1027.539,110.084,-103.989,168.413,46.168,158.626
C08655=1027.545,110.333,-104.009,168.415,46.165,158.626
C08656=1027.550,110.582,-104.028,168.418,46.162,158.626
C08657=1027.556,110.832,-104.047,168.421,46.159,158.626
C08658=1027.562,111.081,-104.067,168.424,46.155,158.625
C08659=1027.568,111.330,-104.086,168.426,46.153,158.625
C08660=1027.574,111.579,-104.106,168.429,46.150,158.625
C08661=1027.580,111.829,-104.126,168.431,46.147,158.625
C08662=1027.587,112.077,-104.145,168.433,46.144,158.624
C08663=1027.592,112.327,-104.165,168.437,46.141,158.624
C08664=1027.598,112.576,-104.185,168.439,46.138,158.624
C08665=1027.604,112.825,-104.204,168.442,46.135,158.623
C08666=1027.610,113.074,-104.224,168.444,46.132,158.623
C08667=1027.616,113.323,-104.243,168.448,46.129,158.623
C08668=1027.621,113.572,-104.264,168.450,46.126,158.622
C08669=1027.627,113.822,-104.283,168.452,46.123,158.622
C08670=1027.633,114.071,-104.303,168.455,46.120,158.622
C08671=1027.639,114.319,-104.323,168.457,46.117,158.622
C08672=1027.645,114.570,-104.342,168.459,46.115,158.621
C08673=1027.651,114.818,-104.362,168.463,46.112,158.621
C08674=1027.656,115.068,-104.383,168.465,46.109,158.621
C08675=1027.662,115.317,-104.402,168.468,46.106,158.621
C08676=1027.668,115.566,-104.422,168.470,46.103,158.620
C08677=1027.674,115.815,-104.442,168.472,46.100,158.620
C08678=1027.680,116.064,-104.461,168.476,46.097,158.620
C08679=1027.686,116.313,-104.481,168.478,46.094,158.620
C08680=1027.691,116.562,-104.502,168.481,46.091,158.619
C08681=1027.697,116.811,-104.521,168.483,46.089,158.619
C08682=1027.703,117.061,-104.541,168.487,46.086,158.619
C08683=1027.709,117.310,-104.561,168.489,46.083,158.619
C08684=1027.715,117.559,-104.581,168.491,46.080,158.618
C08685=1027.721,117.808,-104.601,168.494,46.077,158.618
C08686=1027.726,118.057,-104.621,168.496,46.074,158.618
C08687=1027.732,118.306,-104.641,168.500,46.071,158.617
C08688=1027.739,118.555,-104.661,168.502,46.068,158.617
C08689=1027.744,118.805,-104.681,168.505,46.065,158.617
C08690=1027.750,119.054,-104.701,168.507,46.062,158.617
C08691=1027.756,119.303,-104.721,168.510,46.060,158.616
C08692=1027.762,119.552,-104.741,168.513,46.056,158.616
C08693=1027.768,119.800,-104.761,168.515,46.053,158.616
C08694=1027.774,120.051,-104.781,168.518,46.050,158.616
C08695=1027.780,120.299,-104.801,168.520,46.048,158.615
C08696=1027.786,120.548,-104.821,168.524,46.045,158.615
C08697=1027.791,120.797,-104.841,168.526,46.042,158.615
C08698=1027.797,121.046,-104.861,168.529,46.038,158.614
C08699=1027.803,121.296,-104.881,168.531,46.036,158.614
C08700=1027.809,121.545,-104.901,168.534,46.033,158.614
C08701=1027.815,121.794,-104.921,168.537,46.030,158.614
C08702=1027.821,122.043,-104.941,168.539,46.027,158.613
C08703=1027.827,122.292,-104.961,168.542,46.024,158.613
C08704=1027.833,122.541,-104.981,168.544,46.021,158.613
C08705=1027.839,122.790,-105.001,168.547,46.018,158.612
C08706=1027.845,123.040,-105.021,168.549,46.015,158.612
C08707=1027.850,123.289,-105.041,168.553,46.012,158.612
C08708=1027.857,123.538,-105.062,168.555,46.010,158.612
C08709=1027.864,123.823,-105.084,168.558,46.006,158.611
C08710=1027.870,124.107,-105.108,168.561,46.002,158.611
C08711=1027.878,124.392,-105.130,168.564,45.999,158.611
C08712=1027.884,124.676,-105.153,168.567,45.996,158.610
C08713=1027.890,124.925,-105.173,168.570,45.993,158.610
C08714=1027.897,125.175,-105.194,168.573,45.990,158.610
C08715=1027.903,125.423,-105.214,168.576,45.987,158.609
C08716=1027.908,125.673,-105.234,168.578,45.984,158.609
C08717=1027.914,125.922,-105.255,168.581,45.981,158.609
C08718=1027.920,126.171,-105.275,168.583,45.978,158.609
C08719=1027.926,126.420,-105.295,168.587,45.975,158.608
C08720=1027.932,126.669,-105.314,168.589,45.972,158.608
C08721=1027.938,126.918,-105.335,168.592,45.969,158.608
C08722=1027.944,127.167,-105.355,168.595,45.966,158.608
C08723=1027.950,127.416,-105.375,168.597,45.963,158.607
C08724=1027.957,127.666,-105.396,168.600,45.960,158.607
C08725=1027.963,127.914,-105.416,168.603,45.957,158.607
C08726=1027.968,128.163,-105.436,168.606,45.954,158.606
C08727=1027.975,128.413,-105.456,168.608,45.951,158.606
C08728=1027.981,128.662,-105.476,168.611,45.948,158.606
C08729=1027.987,128.911,-105.497,168.613,45.945,158.606
C08730=1027.992,129.160,-105.517,168.617,45.942,158.605
C08731=1027.998,129.409,-105.537,168.619,45.939,158.605
C08732=1028.005,129.659,-105.558,168.622,45.936,158.605
C08733=1028.011,129.908,-105.578,168.625,45.933,158.604
C08734=1028.017,130.156,-105.598,168.627,45.930,158.604
C08735=1028.023,130.406,-105.618,168.631,45.927,158.604
C08736=1028.029,130.654,-105.639,168.633,45.924,158.604
C08737=1028.035,130.904,-105.660,168.636,45.921,158.603
C08738=1028.041,131.153,-105.680,168.638,45.919,158.603
C08739=1028.046,131.402,-105.701,168.642,45.916,158.603
C08740=1028.053,131.651,-105.722,168.644,45.913,158.603
C08741=1028.058,131.900,-105.742,168.647,45.910,158.602
C08742=1028.064,132.149,-105.763,168.649,45.907,158.602
C08743=1028.070,132.399,-105.783,168.652,45.904,158.602
C08744=1028.076,132.647,-105.804,168.655,45.901,158.601
C08745=1028.082,132.897,-105.825,168.658,45.898,158.601
C08746=1028.088,133.146,-105.845,168.660,45.895,158.601
C08747=1028.094,133.395,-105.865,168.663,45.893,158.601
C08748=1028.100,133.644,-105.887,168.666,45.890,158.600
C08749=1028.106,133.893,-105.907,168.669,45.887,158.600
C08750=1028.111,134.142,-105.927,168.671,45.884,158.600
C08751=1028.117,134.391,-105.949,168.674,45.881,158.600
C08752=1028.123,134.640,-105.969,168.677,45.879,158.599
C08753=1028.129,134.890,-105.990,168.680,45.876,158.599
C08754=1028.135,135.138,-106.010,168.682,45.873,158.599
C08755=1028.141,135.388,-106.031,168.685,45.869,158.599
C08756=1028.148,135.636,-106.052,168.688,45.866,158.598
C08757=1028.153,135.885,-106.073,168.691,45.864,158.598
C08758=1028.159,136.135,-106.093,168.694,45.861,158.598
C08759=1028.165,136.383,-106.114,168.696,45.858,158.598
C08760=1028.171,136.633,-106.135,168.700,45.855,158.597
C08761=1028.177,136.881,-106.156,168.702,45.852,158.597
C08762=1028.183,137.131,-106.177,168.705,45.849,158.597
C08763=1028.188,137.380,-106.197,168.707,45.847,158.597
C08764=1028.195,137.629,-106.218,168.711,45.844,158.596
C08765=1028.200,137.878,-106.239,168.713,45.841,158.596
C08766=1028.207,138.127,-106.261,168.716,45.838,158.596
C08767=1028.213,138.376,-106.280,168.719,45.835,158.596
C08768=1028.219,138.625,-106.302,168.722,45.833,158.595
C08769=1028.224,138.874,-106.323,168.725,45.830,158.595
C08770=1028.231,139.123,-106.344,168.727,45.827,158.595
C08771=1028.236,139.372,-106.364,168.730,45.824,158.595
C08772=1028.242,139.622,-106.386,168.733,45.821,158.594
C08773=1028.249,139.906,-106.410,168.736,45.818,158.594
C08774=1028.255,140.190,-106.433,168.739,45.815,158.594
C08775=1028.261,140.475,-106.458,168.742,45.812,158.594
C08776=1028.269,140.760,-106.482,168.746,45.808,158.593
C08777=1028.274,141.008,-106.503,168.748,45.805,158.593
C08778=1028.281,141.258,-106.524,168.752,45.802,158.593
C08779=1028.286,141.506,-106.545,168.754,45.800,158.592
C08780=1028.293,141.755,-106.567,168.757,45.797,158.592
C08781=1028.298,142.004,-106.587,168.759,45.794,158.592
C08782=1028.304,142.254,-106.609,168.763,45.791,158.592
C08783=1028.309,142.503,-106.629,168.766,45.788,158.591
C08784=1028.316,142.752,-106.650,168.768,45.786,158.591
C08785=1028.322,143.000,-106.672,168.772,45.783,158.591
C08786=1028.328,143.250,-106.693,168.774,45.780,158.591
C08787=1028.334,143.499,-106.714,168.777,45.777,158.590
C08788=1028.339,143.748,-106.736,168.779,45.774,158.590
C08789=1028.346,143.997,-106.757,168.783,45.771,158.590
C08790=1028.352,144.246,-106.777,168.786,45.768,158.590
C08791=1028.358,144.495,-106.799,168.788,45.766,158.589
C08792=1028.363,144.743,-106.820,168.791,45.763,158.589
C08793=1028.369,144.993,-106.842,168.794,45.760,158.589
C08794=1028.375,145.242,-106.863,168.797,45.757,158.589
C08795=1028.381,145.491,-106.884,168.800,45.754,158.588
C08796=1028.388,145.740,-106.905,168.802,45.752,158.588
C08797=1028.393,145.988,-106.926,168.806,45.749,158.588
C08798=1028.399,146.238,-106.947,168.809,45.746,158.588
C08799=1028.405,146.487,-106.969,168.811,45.743,158.587
C08800=1028.411,146.736,-106.990,168.814,45.740,158.587
C08801=1028.417,146.985,-107.012,168.817,45.738,158.587
C08802=1028.423,147.234,-107.033,168.820,45.735,158.587
C08803=1028.429,147.483,-107.055,168.824,45.732,158.587
C08804=1028.435,147.733,-107.075,168.826,45.730,158.586
C08805=1028.440,147.981,-107.097,168.829,45.727,158.586
C08806=1028.446,148.230,-107.118,168.831,45.724,158.586
C08807=1028.453,148.480,-107.140,168.835,45.721,158.586
C08808=1028.458,148.728,-107.161,168.838,45.718,158.585
C08809=1028.464,148.977,-107.183,168.840,45.716,158.585
C08810=1028.470,149.226,-107.204,168.843,45.713,158.585
C08811=1028.476,149.475,-107.226,168.846,45.710,158.585
C08812=1028.482,149.724,-107.247,168.849,45.708,158.585
C08813=1028.487,149.973,-107.269,168.852,45.705,158.584
C08814=1028.493,150.222,-107.291,168.855,45.702,158.584
C08815=1028.499,150.471,-107.313,168.858,45.699,158.584
C08816=1028.505,150.720,-107.334,168.860,45.696,158.584
C08817=1028.511,150.969,-107.355,168.863,45.694,158.583
C08818=1028.517,151.218,-107.377,168.867,45.691,158.583
C08819=1028.523,151.467,-107.398,168.869,45.688,158.583
C08820=1028.529,151.716,-107.420,168.873,45.686,158.583
C08821=1028.535,151.965,-107.442,168.876,45.683,158.582
C08822=1028.540,152.214,-107.464,168.878,45.680,158.582
C08823=1028.546,152.463,-107.485,168.881,45.677,158.582
C08824=1028.552,152.712,-107.507,168.885,45.674,158.582
C08825=1028.558,152.962,-107.528,168.887,45.672,158.581
C08826=1028.564,153.210,-107.550,168.890,45.669,158.581
C08827=1028.570,153.459,-107.572,168.893,45.666,158.581
C08828=1028.577,153.708,-107.594,168.896,45.664,158.581
C08829=1028.581,153.957,-107.616,168.899,45.661,158.581
C08830=1028.588,154.206,-107.637,168.902,45.658,158.580
C08831=1028.594,154.455,-107.659,168.905,45.655,158.580
C08832=1028.600,154.704,-107.680,168.908,45.652,158.580
C08833=1028.605,154.953,-107.703,168.910,45.650,158.580
C08834=1028.611,155.202,-107.725,168.914,45.647,158.580
C08835=1028.617,155.451,-107.746,168.917,45.645,158.579
C08836=1028.623,155.700,-107.768,168.919,45.642,158.579
C08837=1028.630,155.984,-107.793,168.924,45.639,158.579
C08838=1028.636,156.269,-107.818,168.927,45.636,158.579
C08839=1028.643,156.552,-107.843,168.930,45.632,158.578
C08840=1028.650,156.836,-107.868,168.933,45.629,158.578
C08841=1028.656,157.085,-107.890,168.936,45.626,158.578
C08842=1028.662,157.335,-107.912,168.940,45.624,158.578
C08843=1028.668,157.583,-107.934,168.942,45.622,158.577
C08844=1028.674,157.833,-107.956,168.946,45.619,158.577
C08845=1028.679,158.081,-107.977,168.949,45.616,158.577
C08846=1028.686,158.330,-107.999,168.951,45.613,158.577
C08847=1028.691,158.579,-108.022,168.955,45.611,158.577
C08848=1028.697,158.828,-108.044,168.958,45.608,158.576
C08849=1028.704,159.078,-108.065,168.960,45.605,158.576
C08850=1028.710,159.326,-108.087,168.963,45.602,158.576
C08851=1028.715,159.575,-108.109,168.967,45.599,158.576
C08852=1028.721,159.824,-108.132,168.969,45.597,158.576
C08853=1028.727,160.073,-108.154,168.972,45.595,158.575
C08854=1028.733,160.322,-108.177,168.976,45.592,158.575
C08855=1028.737,160.571,-108.199,168.978,45.590,158.575
C08856=1028.744,160.819,-108.221,168.982,45.587,158.575
C08857=1028.749,161.069,-108.243,168.985,45.584,158.575
C08858=1028.755,161.318,-108.266,168.987,45.582,158.574
C08859=1028.760,161.567,-108.289,168.991,45.580,158.574
C08860=1028.766,161.815,-108.311,168.994,45.577,158.574
C08861=1028.772,162.064,-108.334,168.997,45.575,158.574
C08862=1028.777,162.314,-108.356,169.000,45.572,158.574
C08863=1028.784,162.562,-108.378,169.003,45.569,158.573
C08864=1028.789,162.812,-108.400,169.006,45.567,158.573
C08865=1028.794,163.060,-108.423,169.009,45.564,158.573
C08866=1028.800,163.309,-108.446,169.013,45.562,158.573
C08867=1028.806,163.558,-108.467,169.015,45.559,158.573
C08868=1028.812,163.807,-108.490,169.018,45.556,158.572
C08869=1028.818,164.056,-108.513,169.022,45.554,158.572
C08870=1028.824,164.305,-108.535,169.024,45.551,158.572
C08871=1028.830,164.554,-108.558,169.027,45.549,158.572
C08872=1028.835,164.802,-108.581,169.031,45.546,158.572
C08873=1028.840,165.052,-108.603,169.033,45.544,158.572
C08874=1028.847,165.300,-108.625,169.037,45.541,158.571
C08875=1028.852,165.549,-108.648,169.040,45.538,158.571
C08876=1028.858,165.799,-108.670,169.043,45.536,158.571
C08877=1028.864,166.048,-108.693,169.046,45.533,158.571
C08878=1028.870,166.296,-108.716,169.049,45.531,158.571
C08879=1028.876,166.545,-108.739,169.052,45.528,158.571
C08880=1028.881,166.795,-108.761,169.055,45.526,158.570
C08881=1028.888,167.043,-108.783,169.058,45.523,158.570
C08882=1028.893,167.291,-108.806,169.062,45.521,158.570
C08883=1028.899,167.540,-108.829,169.065,45.518,158.570
C08884=1028.904,167.790,-108.851,169.067,45.516,158.570
C08885=1028.910,168.038,-108.873,169.071,45.513,158.570
C08886=1028.916,168.287,-108.896,169.074,45.511,158.569
C08887=1028.922,168.536,-108.919,169.077,45.508,158.569
C08888=1028.928,168.785,-108.942,169.080,45.506,158.569
C08889=1028.934,169.034,-108.964,169.083,45.503,158.569
C08890=1028.940,169.283,-108.987,169.087,45.501,158.569
C08891=1028.945,169.532,-109.010,169.090,45.498,158.568
C08892=1028.951,169.781,-109.033,169.093,45.496,158.568
C08893=1028.958,170.030,-109.055,169.096,45.493,158.568
C08894=1028.963,170.278,-109.078,169.099,45.490,158.568
C08895=1028.969,170.527,-109.101,169.103,45.488,158.568
C08896=1028.975,170.776,-109.124,169.106,45.485,158.567
C08897=1028.981,171.025,-109.145,169.109,45.483,158.567
C08898=1028.987,171.274,-109.168,169.112,45.480,158.567
C08899=1028.992,171.523,-109.191,169.115,45.478,158.567
C08900=1028.998,171.772,-109.214,169.119,45.475,158.567
C08901=1029.005,172.056,-109.241,169.122,45.472,158.567
C08902=1029.012,172.340,-109.266,169.125,45.469,158.566
C08903=1029.019,172.624,-109.292,169.129,45.466,158.566
C08904=1029.025,172.907,-109.318,169.133,45.463,158.566
C08905=1029.031,173.156,-109.341,169.136,45.461,158.566
C08906=1029.038,173.404,-109.364,169.140,45.458,158.566
C08907=1029.043,173.653,-109.387,169.143,45.456,158.566
C08908=1029.050,173.903,-109.410,169.145,45.453,158.565
C08909=1029.055,174.152,-109.433,169.149,45.451,158.565
C08910=1029.062,174.400,-109.455,169.152,45.448,158.565
C08911=1029.068,174.649,-109.478,169.156,45.446,158.565
C08912=1029.073,174.898,-109.501,169.159,45.443,158.565
C08913=1029.079,175.147,-109.524,169.162,45.440,158.564
C08914=1029.085,175.396,-109.547,169.165,45.438,158.564
C08915=1029.091,175.644,-109.569,169.168,45.435,158.564
C08916=1029.097,175.893,-109.592,169.172,45.433,158.564
C08917=1029.103,176.143,-109.616,169.175,45.430,158.564
C08918=1029.109,176.392,-109.639,169.179,45.428,158.564
C08919=1029.115,176.640,-109.661,169.182,45.425,158.563
C08920=1029.121,176.889,-109.684,169.185,45.423,158.563
C08921=1029.127,177.137,-109.707,169.189,45.420,158.563
C08922=1029.133,177.386,-109.730,169.191,45.418,158.563
C08923=1029.139,177.636,-109.754,169.194,45.415,158.563
C08924=1029.146,177.885,-109.776,169.198,45.412,158.562
C08925=1029.151,178.133,-109.799,169.201,45.410,158.562
C08926=1029.157,178.382,-109.822,169.205,45.407,158.562
C08927=1029.163,178.631,-109.846,169.208,45.405,158.562
C08928=1029.170,178.880,-109.869,169.211,45.402,158.562
C08929=1029.176,179.129,-109.891,169.215,45.400,158.562
C08930=1029.182,179.378,-109.914,169.218,45.397,158.561
C08931=1029.187,179.627,-109.937,169.222,45.394,158.561
C08932=1029.194,179.876,-109.961,169.225,45.392,158.561
C08933=1029.200,180.124,-109.984,169.228,45.390,158.561
C08934=1029.206,180.373,-110.007,169.231,45.387,158.561
C08935=1029.212,180.622,-110.029,169.234,45.385,158.561
C08936=1029.219,180.871,-110.053,169.238,45.382,158.560
C08937=1029.224,181.120,-110.076,169.241,45.379,158.560
C08938=1029.230,181.369,-110.099,169.244,45.377,158.560
C08939=1029.237,181.617,-110.122,169.248,45.374,158.560
C08940=1029.243,181.866,-110.146,169.251,45.371,158.560
C08941=1029.249,182.115,-110.169,169.255,45.369,158.560
C08942=1029.255,182.364,-110.192,169.258,45.366,158.560
C08943=1029.261,182.613,-110.216,169.262,45.364,158.559
C08944=1029.268,182.862,-110.238,169.265,45.361,158.559
C08945=1029.273,183.110,-110.262,169.268,45.359,158.559
C08946=1029.279,183.359,-110.285,169.272,45.357,158.559
C08947=1029.284,183.608,-110.309,169.276,45.355,158.559
C08948=1029.290,183.857,-110.333,169.278,45.352,158.559
C08949=1029.297,184.106,-110.356,169.281,45.350,158.559
C08950=1029.302,184.354,-110.381,169.285,45.348,158.559
C08951=1029.308,184.603,-110.404,169.288,45.345,158.558
C08952=1029.313,184.852,-110.428,169.292,45.343,158.558
C08953=1029.320,185.101,-110.452,169.296,45.341,158.558
C08954=1029.325,185.350,-110.475,169.299,45.338,158.558
C08955=1029.331,185.598,-110.499,169.302,45.336,158.558
C08956=1029.337,185.848,-110.522,169.305,45.334,158.558
C08957=1029.342,186.096,-110.547,169.308,45.332,158.558
C08958=1029.348,186.345,-110.570,169.312,45.329,158.558
C08959=1029.354,186.594,-110.595,169.315,45.327,158.557
C08960=1029.360,186.843,-110.618,169.319,45.324,158.557
C08961=1029.366,187.091,-110.642,169.322,45.322,158.557
C08962=1029.371,187.340,-110.666,169.326,45.320,158.557
C08963=1029.377,187.589,-110.689,169.329,45.318,158.557
C08964=1029.383,187.838,-110.713,169.333,45.316,158.557
C08965=1029.390,188.121,-110.741,169.336,45.313,158.557
C08966=1029.396,188.404,-110.768,169.341,45.310,158.557
C08967=1029.403,188.688,-110.795,169.344,45.307,158.556
C08968=1029.410,188.971,-110.822,169.349,45.305,158.556
C08969=1029.416,189.220,-110.846,169.352,45.303,158.556
C08970=1029.422,189.468,-110.870,169.356,45.301,158.556
C08971=1029.427,189.718,-110.894,169.359,45.298,158.556
C08972=1029.433,189.966,-110.917,169.363,45.295,158.556
C08973=1029.439,190.215,-110.942,169.366,45.293,158.556
C08974=1029.445,190.464,-110.966,169.370,45.291,158.556
C08975=1029.451,190.712,-110.990,169.373,45.289,158.556
C08976=1029.457,190.961,-111.014,169.376,45.287,158.556
C08977=1029.463,191.210,-111.038,169.379,45.285,158.555
C08978=1029.469,191.459,-111.062,169.383,45.282,158.555
C08979=1029.475,191.708,-111.085,169.386,45.280,158.555
C08980=1029.480,191.956,-111.110,169.390,45.277,158.555
C08981=1029.487,192.205,-111.134,169.393,45.275,158.555
C08982=1029.492,192.454,-111.158,169.397,45.273,158.555
C08983=1029.499,192.703,-111.182,169.400,45.271,158.555
C08984=1029.505,192.951,-111.205,169.405,45.268,158.555
C08985=1029.511,193.200,-111.230,169.408,45.266,158.555
C08986=1029.517,193.449,-111.254,169.412,45.264,158.555
C08987=1029.523,193.698,-111.278,169.416,45.262,158.555
C08988=1029.529,193.946,-111.302,169.419,45.260,158.554
C08989=1029.535,194.196,-111.327,169.422,45.257,158.554
C08990=1029.541,194.444,-111.350,169.426,45.255,158.554
